LIN {X 0,Y 310.532,Z 504.322,A -85,B 0,C 180,E1 -15911.191,E2 -15911.191} C_VEL
LIN {X 0,Y 308.815,Z 514.48,A -85,B 0,C 180,E1 -15912.908,E2 -15912.908} C_VEL
LIN {X 0,Y 307.317,Z 523.179,A -85,B 0,C 180,E1 -15914.758,E2 -15914.758} C_VEL
LIN {X 0,Y 305.943,Z 530.654,A -85,B 0,C 180,E1 -15916.725,E2 -15916.725} C_VEL
LIN {X 0,Y 304.932,Z 536.676,A -85,B 0,C 180,E1 -15918.708,E2 -15918.708} C_VEL
LIN {X 0,Y 304.258,Z 541.45,A -85,B 0,C 180,E1 -15920.7,E2 -15920.7} C_VEL
LIN {X 0,Y 303.838,Z 545.114,A -85,B 0,C 180,E1 -15922.696,E2 -15922.696} C_VEL
LIN {X 0,Y 303.635,Z 547.768,A -85,B 0,C 180,E1 -15924.692,E2 -15924.692} C_VEL
LIN {X 0,Y 303.631,Z 549.032,A -85,B 0,C 180,E1 -15926.023,E2 -15926.023} C_VEL
LIN {X 0,Y 303.623,Z 549.85,A -85,B 0,C 180,E1 -15927.351,E2 -15927.351} C_VEL
LIN {X 0,Y 303.613,Z 550.259,A -85,B 0,C 180,E1 -15928.678,E2 -15928.678} C_VEL
LIN {X 0,Y 303.669,Z 550.277,A -85,B 0,C 180,E1 -15930.004,E2 -15930.004} C_VEL
LIN {X 0,Y 303.626,Z 549.898,A -85,B 0,C 180,E1 -15931.331,E2 -15931.331} C_VEL
LIN {X 0,Y 303.63,Z 549.077,A -85,B 0,C 180,E1 -15932.657,E2 -15932.657} C_VEL
LIN {X 0,Y 303.652,Z 547.834,A -85,B 0,C 180,E1 -15933.986,E2 -15933.986} C_VEL
LIN {X 0,Y 303.625,Z 545.862,A -85,B 0,C 180,E1 -15935.544,E2 -15935.544} C_VEL
LIN {X 0,Y 303.837,Z 542.819,A -85,B 0,C 180,E1 -15937.313,E2 -15937.313} C_VEL
LIN {X 0,Y 304.202,Z 538.362,A -85,B 0,C 180,E1 -15939.311,E2 -15939.311} C_VEL
LIN {X 0,Y 304.78,Z 532.679,A -85,B 0,C 180,E1 -15941.307,E2 -15941.307} C_VEL
LIN {X 0,Y 305.726,Z 525.55,A -85,B 0,C 180,E1 -15943.293,E2 -15943.293} C_VEL
LIN {X 0,Y 306.996,Z 516.63,A -85,B 0,C 180,E1 -15945.267,E2 -15945.267} C_VEL
LIN {X 0,Y 308.203,Z 507.257,A -85,B 0,C 180,E1 -15946.943,E2 -15946.943} C_VEL
LIN {X 0,Y 309.424,Z 497.348,A -85,B 0,C 180,E1 -15948.373,E2 -15948.373} C_VEL
LIN {X 0,Y 310.841,Z 486.113,A -85,B 0,C 180,E1 -15949.656,E2 -15949.656} C_VEL
LIN {X 0,Y 312.223,Z 473.536,A -85,B 0,C 180,E1 -15950.767,E2 -15950.767} C_VEL
LIN {X 0,Y 313.349,Z 460.657,A -85,B 0,C 180,E1 -15951.593,E2 -15951.593} C_VEL
LIN {X 0,Y 314.132,Z 448.168,A -85,B 0,C 180,E1 -15952.141,E2 -15952.141} C_VEL
LIN {X 0,Y 314.99,Z 419.656,A -85,B 0,C 180,E1 -15952.858,E2 -15952.858} C_VEL
LIN {X 0,Y 315.888,Z 380.038,A -85,B 0,C 180,E1 -15953.803,E2 -15953.803} C_VEL
LIN {X 0,Y 310.923,Z 346.154,A -85,B 0,C 180,E1 -15955.03,E2 -15955.03} C_VEL
LIN {X 0,Y 309.644,Z 338.018,A -85,B 0,C 180,E1 -15955.349,E2 -15955.349} C_VEL
LIN {X 0,Y 309.994,Z 334.693,A -85,B 0,C 180,E1 -15956.24,E2 -15956.24} C_VEL
LIN {X 0,Y 308.58,Z 326.696,A -85,B 0,C 180,E1 -15958.576,E2 -15958.576} C_VEL
LIN {X 0,Y 305.968,Z 314.569,A -85,B 0,C 180,E1 -15962.281,E2 -15962.281} C_VEL
LIN {X 0,Y 305.501,Z 312.43,A -85,B 0,C 180,E1 -15963.022,E2 -15963.022} C_VEL
LIN {X 0,Y 305.481,Z 312.431,A -85,B 0,C 180,E1 -15966.741,E2 -15966.741} C_VEL
LIN {X 0,Y 305.46,Z 312.438,A -85,B 0,C 180,E1 -15970.601,E2 -15970.601} C_VEL
LIN {X 0,Y 305.431,Z 312.437,A -85,B 0,C 180,E1 -15973.656,E2 -15973.656} C_VEL
LIN {X 0,Y 305.459,Z 312.433,A -85,B 0,C 180,E1 -15977.415,E2 -15977.415} C_VEL
LIN {X 0,Y 305.471,Z 312.431,A -85,B 0,C 180,E1 -15981.597,E2 -15981.597} C_VEL
LIN {X 0,Y 305.466,Z 312.435,A -85,B 0,C 180,E1 -15984.887,E2 -15984.887} C_VEL
LIN {X 0,Y 305.446,Z 312.437,A -85,B 0,C 180,E1 -15988.359,E2 -15988.359} C_VEL
LIN {X 0,Y 305.509,Z 312.43,A -85,B 0,C 180,E1 -15991.113,E2 -15991.113} C_VEL
LIN {X 0,Y 305.567,Z 312.419,A -85,B 0,C 180,E1 -15994.087,E2 -15994.087} C_VEL
LIN {X 0,Y 305.465,Z 312.433,A -85,B 0,C 180,E1 -15998.4,E2 -15998.4} C_VEL
LIN {X 0,Y 305.535,Z 312.42,A -85,B 0,C 180,E1 -16002.601,E2 -16002.601} C_VEL
LIN {X 0,Y 305.626,Z 312.412,A -85,B 0,C 180,E1 -16005.348,E2 -16005.348} C_VEL
LIN {X 0,Y 305.624,Z 312.416,A -85,B 0,C 180,E1 -16009.399,E2 -16009.399} C_VEL
LIN {X 0,Y 305.787,Z 312.391,A -85,B 0,C 180,E1 -16012.074,E2 -16012.074} C_VEL
LIN {X 0,Y 305.68,Z 312.402,A -85,B 0,C 180,E1 -16014.723,E2 -16014.723} C_VEL
LIN {X 0,Y 305.952,Z 312.362,A -85,B 0,C 180,E1 -16018.684,E2 -16018.684} C_VEL
LIN {X 0,Y 305.951,Z 312.37,A -85,B 0,C 180,E1 -16021.316,E2 -16021.316} C_VEL
LIN {X 0,Y 305.665,Z 312.409,A -85,B 0,C 180,E1 -16025.277,E2 -16025.277} C_VEL
LIN {X 0,Y 305.738,Z 312.4,A -85,B 0,C 180,E1 -16027.928,E2 -16027.928} C_VEL
LIN {X 0,Y 305.596,Z 312.419,A -85,B 0,C 180,E1 -16031.945,E2 -16031.945} C_VEL
LIN {X 0,Y 305.609,Z 312.414,A -85,B 0,C 180,E1 -16035.013,E2 -16035.013} C_VEL
LIN {X 0,Y 305.518,Z 312.422,A -85,B 0,C 180,E1 -16038.787,E2 -16038.787} C_VEL
LIN {X 0,Y 305.459,Z 312.432,A -85,B 0,C 180,E1 -16043.025,E2 -16043.025} C_VEL
LIN {X 0,Y 305.445,Z 312.437,A -85,B 0,C 180,E1 -16046.186,E2 -16046.186} C_VEL
LIN {X 0,Y 305.423,Z 312.431,A -85,B 0,C 180,E1 -16049.023,E2 -16049.023} C_VEL
LIN {X 0,Y 305.437,Z 312.427,A -85,B 0,C 180,E1 -16051.953,E2 -16051.953} C_VEL
LIN {X 0,Y 305.463,Z 312.429,A -85,B 0,C 180,E1 -16055.113,E2 -16055.113} C_VEL
LIN {X 0,Y 305.438,Z 312.44,A -85,B 0,C 180,E1 -16058.524,E2 -16058.524} C_VEL
LIN {X 0,Y 305.406,Z 312.442,A -85,B 0,C 180,E1 -16062.574,E2 -16062.574} C_VEL
LIN {X 0,Y 305.42,Z 312.441,A -85,B 0,C 180,E1 -16066.342,E2 -16066.342} C_VEL
LIN {X 0,Y 305.396,Z 312.439,A -85,B 0,C 180,E1 -16069.88,E2 -16069.88} C_VEL
LIN {X 0,Y 305.452,Z 312.433,A -85,B 0,C 180,E1 -16073.639,E2 -16073.639} C_VEL
LIN {X 0,Y 305.448,Z 312.435,A -85,B 0,C 180,E1 -16076.479,E2 -16076.479} C_VEL
LIN {X 0,Y 305.418,Z 312.439,A -85,B 0,C 180,E1 -16079.583,E2 -16079.583} C_VEL
LIN {X 0,Y 305.459,Z 312.435,A -85,B 0,C 180,E1 -16082.6,E2 -16082.6} C_VEL
LIN {X 0,Y 305.479,Z 312.431,A -85,B 0,C 180,E1 -16085.533,E2 -16085.533} C_VEL
LIN {X 0,Y 305.49,Z 312.43,A -85,B 0,C 180,E1 -16089.81,E2 -16089.81} C_VEL
LIN {X 0,Y 305.557,Z 312.421,A -85,B 0,C 180,E1 -16093.975,E2 -16093.975} C_VEL
LIN {X 0,Y 305.592,Z 312.417,A -85,B 0,C 180,E1 -16096.701,E2 -16096.701} C_VEL
LIN {X 0,Y 305.758,Z 312.399,A -85,B 0,C 180,E1 -16101.258,E2 -16101.258} C_VEL
LIN {X 0,Y 305.789,Z 312.396,A -85,B 0,C 180,E1 -16103.397,E2 -16103.397} C_VEL
LIN {X 0,Y 305.948,Z 312.372,A -85,B 0,C 180,E1 -16108.68,E2 -16108.68} C_VEL
LIN {X 0,Y 305.937,Z 312.375,A -85,B 0,C 180,E1 -16111.312,E2 -16111.312} C_VEL
LIN {X 0,Y 305.675,Z 312.496,A -85,B 0,C 180,E1 -16115.065,E2 -16115.065} C_VEL
LIN {X 0,Y 306.684,Z 317.033,A -85,B 0,C 180,E1 -16116.513,E2 -16116.513} C_VEL
LIN {X 0,Y 315.207,Z 340.384,A -85,B 0,C 180,E1 -16117.762,E2 -16117.762} C_VEL
LIN {X 0,Y 316.534,Z 347.221,A -85,B 0,C 180,E1 -16118.031,E2 -16118.031} C_VEL
LIN {X 0,Y 314.507,Z 424.142,A -85,B 0,C 180,E1 -16119.877,E2 -16119.877} C_VEL
LIN {X 0,Y 313.857,Z 437.197,A -85,B 0,C 180,E1 -16120.437,E2 -16120.437} C_VEL
LIN {X 0,Y 312.968,Z 449.965,A -85,B 0,C 180,E1 -16121.245,E2 -16121.245} C_VEL
LIN {X 0,Y 311.97,Z 461.032,A -85,B 0,C 180,E1 -16122.187,E2 -16122.187} C_VEL
LIN {X 0,Y 310.666,Z 472.181,A -85,B 0,C 180,E1 -16123.402,E2 -16123.402} C_VEL
LIN {X 0,Y 309.211,Z 483.594,A -85,B 0,C 180,E1 -16124.978,E2 -16124.978} C_VEL
LIN {X 0,Y 308.01,Z 492.9,A -85,B 0,C 180,E1 -16126.597,E2 -16126.597} C_VEL
LIN {X 0,Y 306.843,Z 501.093,A -85,B 0,C 180,E1 -16128.351,E2 -16128.351} C_VEL
LIN {X 0,Y 305.759,Z 509.186,A -85,B 0,C 180,E1 -16130.514,E2 -16130.514} C_VEL
LIN {X 0,Y 305.129,Z 514.182,A -85,B 0,C 180,E1 -16132.188,E2 -16132.188} C_VEL
LIN {X 0,Y 304.432,Z 519.747,A -85,B 0,C 180,E1 -16134.547,E2 -16134.547} C_VEL
LIN {X 0,Y 303.886,Z 523.579,A -85,B 0,C 180,E1 -16136.8,E2 -16136.8} C_VEL
LIN {X 0,Y 303.543,Z 526.171,A -85,B 0,C 180,E1 -16139.085,E2 -16139.085} C_VEL
LIN {X 0,Y 303.425,Z 527.406,A -85,B 0,C 180,E1 -16141.018,E2 -16141.018} C_VEL
LIN {X 0,Y 303.471,Z 527.743,A -85,B 0,C 180,E1 -16143.517,E2 -16143.517} C_VEL
LIN {X 0,Y 303.709,Z 526.753,A -85,B 0,C 180,E1 -16145.912,E2 -16145.912} C_VEL
LIN {X 0,Y 304.143,Z 524.521,A -85,B 0,C 180,E1 -16148.218,E2 -16148.218} C_VEL
LIN {X 0,Y 304.8,Z 521.115,A -85,B 0,C 180,E1 -16150.456,E2 -16150.456} C_VEL
LIN {X 0,Y 305.637,Z 516.547,A -85,B 0,C 180,E1 -16152.623,E2 -16152.623} C_VEL
LIN {X 0,Y 306.766,Z 510.68,A -85,B 0,C 180,E1 -16154.748,E2 -16154.748} C_VEL
LIN {X 0,Y 308.203,Z 503.227,A -85,B 0,C 180,E1 -16156.851,E2 -16156.851} C_VEL
LIN {X 0,Y 309.972,Z 493.999,A -85,B 0,C 180,E1 -16158.889,E2 -16158.889} C_VEL
LIN {X 0,Y 311.555,Z 484.866,A -85,B 0,C 180,E1 -16160.507,E2 -16160.507} C_VEL
LIN {X 0,Y 312.9,Z 475.839,A -85,B 0,C 180,E1 -16161.814,E2 -16161.814} C_VEL
LIN {X 0,Y 314.575,Z 464.879,A -85,B 0,C 180,E1 -16163.071,E2 -16163.071} C_VEL
LIN {X 0,Y 315.779,Z 454.371,A -85,B 0,C 180,E1 -16164.041,E2 -16164.041} C_VEL
LIN {X 0,Y 316.943,Z 441.922,A -85,B 0,C 180,E1 -16164.915,E2 -16164.915} C_VEL
LIN {X 0,Y 317.748,Z 429.439,A -85,B 0,C 180,E1 -16165.534,E2 -16165.534} C_VEL
LIN {X 0,Y 317.977,Z 425.769,A -85,B 0,C 180,E1 -16165.662,E2 -16165.662} C_VEL
LIN {X 0,Y 317.615,Z 420.025,A -85,B 0,C 180,E1 -16165.907,E2 -16165.907} C_VEL
LIN {X 0,Y 313.109,Z 401.411,A -85,B 0,C 180,E1 -16166.843,E2 -16166.843} C_VEL
LIN {X 0,Y 312.707,Z 395.612,A -85,B 0,C 180,E1 -16167.035,E2 -16167.035} C_VEL
LIN {X 0,Y 314.177,Z 349.617,A -85,B 0,C 180,E1 -16168.164,E2 -16168.164} C_VEL
LIN {X 0,Y 308.843,Z 336.559,A -85,B 0,C 180,E1 -16169.123,E2 -16169.123} C_VEL
LIN {X 0,Y 301.142,Z 320.791,A -85,B 0,C 180,E1 -16170.507,E2 -16170.507} C_VEL
LIN {X 0,Y 299.59,Z 317.573,A -85,B 0,C 180,E1 -16170.823,E2 -16170.823} C_VEL
LIN {X 0,Y 298.45,Z 313.316,A -85,B 0,C 180,E1 -16172.38,E2 -16172.38} C_VEL
LIN {X 0,Y 298.445,Z 313.316,A -85,B 0,C 180,E1 -16174.92,E2 -16174.92} C_VEL
LIN {X 0,Y 298.397,Z 313.319,A -85,B 0,C 180,E1 -16179.311,E2 -16179.311} C_VEL
LIN {X 0,Y 298.491,Z 313.306,A -85,B 0,C 180,E1 -16182.176,E2 -16182.176} C_VEL
LIN {X 0,Y 298.545,Z 313.299,A -85,B 0,C 180,E1 -16184.992,E2 -16184.992} C_VEL
LIN {X 0,Y 298.539,Z 313.292,A -85,B 0,C 180,E1 -16189.145,E2 -16189.145} C_VEL
LIN {X 0,Y 298.688,Z 313.277,A -85,B 0,C 180,E1 -16191.884,E2 -16191.884} C_VEL
LIN {X 0,Y 298.611,Z 313.29,A -85,B 0,C 180,E1 -16194.598,E2 -16194.598} C_VEL
LIN {X 0,Y 298.879,Z 313.252,A -85,B 0,C 180,E1 -16198.653,E2 -16198.653} C_VEL
LIN {X 0,Y 298.879,Z 313.255,A -85,B 0,C 180,E1 -16201.347,E2 -16201.347} C_VEL
LIN {X 0,Y 298.745,Z 313.268,A -85,B 0,C 180,E1 -16206.755,E2 -16206.755} C_VEL
LIN {X 0,Y 298.638,Z 313.286,A -85,B 0,C 180,E1 -16209.482,E2 -16209.482} C_VEL
LIN {X 0,Y 298.507,Z 313.301,A -85,B 0,C 180,E1 -16213.617,E2 -16213.617} C_VEL
LIN {X 0,Y 298.504,Z 313.29,A -85,B 0,C 180,E1 -16216.411,E2 -16216.411} C_VEL
LIN {X 0,Y 298.494,Z 313.293,A -85,B 0,C 180,E1 -16219.669,E2 -16219.669} C_VEL
LIN {X 0,Y 298.437,Z 313.301,A -85,B 0,C 180,E1 -16223.599,E2 -16223.599} C_VEL
LIN {X 0,Y 298.453,Z 313.305,A -85,B 0,C 180,E1 -16226.578,E2 -16226.578} C_VEL
LIN {X 0,Y 298.384,Z 313.315,A -85,B 0,C 180,E1 -16229.645,E2 -16229.645} C_VEL
LIN {X 0,Y 298.362,Z 313.316,A -85,B 0,C 180,E1 -16232.804,E2 -16232.804} C_VEL
LIN {X 0,Y 298.457,Z 313.308,A -85,B 0,C 180,E1 -16236.823,E2 -16236.823} C_VEL
LIN {X 0,Y 298.428,Z 313.311,A -85,B 0,C 180,E1 -16241.108,E2 -16241.108} C_VEL
LIN {X 0,Y 298.463,Z 313.314,A -85,B 0,C 180,E1 -16245.066,E2 -16245.066} C_VEL
LIN {X 0,Y 298.43,Z 313.315,A -85,B 0,C 180,E1 -16248.903,E2 -16248.903} C_VEL
LIN {X 0,Y 298.449,Z 313.306,A -85,B 0,C 180,E1 -16253.192,E2 -16253.192} C_VEL
LIN {X 0,Y 298.453,Z 313.458,A -85,B 0,C 180,E1 -16254.395,E2 -16254.395} C_VEL
LIN {X 0,Y 301.098,Z 323.779,A -85,B 0,C 180,E1 -16257.934,E2 -16257.934} C_VEL
LIN {X 0,Y 303.507,Z 334.535,A -85,B 0,C 180,E1 -16261.363,E2 -16261.363} C_VEL
LIN {X 0,Y 303.784,Z 335.948,A -85,B 0,C 180,E1 -16261.77,E2 -16261.77} C_VEL
LIN {X 0,Y 306.903,Z 343.742,A -85,B 0,C 180,E1 -16262.363,E2 -16262.363} C_VEL
LIN {X 0,Y 311.12,Z 366.166,A -85,B 0,C 180,E1 -16263.476,E2 -16263.476} C_VEL
LIN {X 0,Y 313.3,Z 382.701,A -85,B 0,C 180,E1 -16264.165,E2 -16264.165} C_VEL
LIN {X 0,Y 311.187,Z 445.435,A -85,B 0,C 180,E1 -16265.72,E2 -16265.72} C_VEL
LIN {X 0,Y 310.209,Z 458.829,A -85,B 0,C 180,E1 -16266.294,E2 -16266.294} C_VEL
LIN {X 0,Y 308.892,Z 471.237,A -85,B 0,C 180,E1 -16267.075,E2 -16267.075} C_VEL
LIN {X 0,Y 307.374,Z 482.408,A -85,B 0,C 180,E1 -16268.018,E2 -16268.018} C_VEL
LIN {X 0,Y 305.621,Z 494.017,A -85,B 0,C 180,E1 -16269.301,E2 -16269.301} C_VEL
LIN {X 0,Y 303.838,Z 504.506,A -85,B 0,C 180,E1 -16270.761,E2 -16270.761} C_VEL
LIN {X 0,Y 302.116,Z 514.002,A -85,B 0,C 180,E1 -16272.403,E2 -16272.403} C_VEL
LIN {X 0,Y 300.442,Z 523.19,A -85,B 0,C 180,E1 -16274.4,E2 -16274.4} C_VEL
LIN {X 0,Y 299.009,Z 530.619,A -85,B 0,C 180,E1 -16276.411,E2 -16276.411} C_VEL
LIN {X 0,Y 297.924,Z 536.598,A -85,B 0,C 180,E1 -16278.438,E2 -16278.438} C_VEL
LIN {X 0,Y 297.229,Z 541.333,A -85,B 0,C 180,E1 -16280.478,E2 -16280.478} C_VEL
LIN {X 0,Y 296.786,Z 544.96,A -85,B 0,C 180,E1 -16282.521,E2 -16282.521} C_VEL
LIN {X 0,Y 296.55,Z 547.576,A -85,B 0,C 180,E1 -16284.565,E2 -16284.565} C_VEL
LIN {X 0,Y 296.528,Z 548.815,A -85,B 0,C 180,E1 -16285.927,E2 -16285.927} C_VEL
LIN {X 0,Y 296.548,Z 549.607,A -85,B 0,C 180,E1 -16287.288,E2 -16287.288} C_VEL
LIN {X 0,Y 296.53,Z 550,A -85,B 0,C 180,E1 -16288.646,E2 -16288.646} C_VEL
LIN {X 0,Y 296.581,Z 550.004,A -85,B 0,C 180,E1 -16290.004,E2 -16290.004} C_VEL
LIN {X 0,Y 296.542,Z 549.604,A -85,B 0,C 180,E1 -16291.362,E2 -16291.362} C_VEL
LIN {X 0,Y 296.555,Z 548.757,A -85,B 0,C 180,E1 -16292.721,E2 -16292.721} C_VEL
LIN {X 0,Y 296.566,Z 547.498,A -85,B 0,C 180,E1 -16294.081,E2 -16294.081} C_VEL
LIN {X 0,Y 296.574,Z 544.796,A -85,B 0,C 180,E1 -16296.125,E2 -16296.125} C_VEL
LIN {X 0,Y 296.878,Z 541.05,A -85,B 0,C 180,E1 -16298.17,E2 -16298.17} C_VEL
LIN {X 0,Y 297.346,Z 536.154,A -85,B 0,C 180,E1 -16300.214,E2 -16300.214} C_VEL
LIN {X 0,Y 298.049,Z 529.959,A -85,B 0,C 180,E1 -16302.256,E2 -16302.256} C_VEL
LIN {X 0,Y 299.19,Z 522.25,A -85,B 0,C 180,E1 -16304.283,E2 -16304.283} C_VEL
LIN {X 0,Y 300.333,Z 514.337,A -85,B 0,C 180,E1 -16305.963,E2 -16305.963} C_VEL
LIN {X 0,Y 301.559,Z 504.648,A -85,B 0,C 180,E1 -16307.639,E2 -16307.639} C_VEL
LIN {X 0,Y 303.043,Z 493.923,A -85,B 0,C 180,E1 -16309.125,E2 -16309.125} C_VEL
LIN {X 0,Y 304.318,Z 483.564,A -85,B 0,C 180,E1 -16310.271,E2 -16310.271} C_VEL
LIN {X 0,Y 305.655,Z 471.217,A -85,B 0,C 180,E1 -16311.323,E2 -16311.323} C_VEL
LIN {X 0,Y 306.839,Z 457.559,A -85,B 0,C 180,E1 -16312.164,E2 -16312.164} C_VEL
LIN {X 0,Y 307.587,Z 444.598,A -85,B 0,C 180,E1 -16312.682,E2 -16312.682} C_VEL
LIN {X 0,Y 309.249,Z 381.078,A -85,B 0,C 180,E1 -16314.236,E2 -16314.236} C_VEL
LIN {X 0,Y 304.445,Z 347.745,A -85,B 0,C 180,E1 -16315.47,E2 -16315.47} C_VEL
LIN {X 0,Y 302.859,Z 337.766,A -85,B 0,C 180,E1 -16315.876,E2 -16315.876} C_VEL
LIN {X 0,Y 302.829,Z 334.116,A -85,B 0,C 180,E1 -16316.91,E2 -16316.91} C_VEL
LIN {X 0,Y 300.678,Z 323.498,A -85,B 0,C 180,E1 -16320.136,E2 -16320.136} C_VEL
LIN {X 0,Y 298.446,Z 313.31,A -85,B 0,C 180,E1 -16323.401,E2 -16323.401} C_VEL
LIN {X 0,Y 298.452,Z 313.307,A -85,B 0,C 180,E1 -16326.809,E2 -16326.809} C_VEL
LIN {X 0,Y 298.393,Z 313.316,A -85,B 0,C 180,E1 -16331.089,E2 -16331.089} C_VEL
LIN {X 0,Y 298.405,Z 313.312,A -85,B 0,C 180,E1 -16333.104,E2 -16333.104} C_VEL
LIN {X 0,Y 298.409,Z 313.314,A -85,B 0,C 180,E1 -16336.922,E2 -16336.922} C_VEL
LIN {X 0,Y 298.403,Z 313.314,A -85,B 0,C 180,E1 -16341.009,E2 -16341.009} C_VEL
LIN {X 0,Y 298.41,Z 313.312,A -85,B 0,C 180,E1 -16343.929,E2 -16343.929} C_VEL
LIN {X 0,Y 298.397,Z 313.315,A -85,B 0,C 180,E1 -16347.2,E2 -16347.2} C_VEL
LIN {X 0,Y 298.457,Z 313.305,A -85,B 0,C 180,E1 -16351.904,E2 -16351.904} C_VEL
LIN {X 0,Y 298.484,Z 313.305,A -85,B 0,C 180,E1 -16354.924,E2 -16354.924} C_VEL
LIN {X 0,Y 298.42,Z 313.311,A -85,B 0,C 180,E1 -16359.313,E2 -16359.313} C_VEL
LIN {X 0,Y 298.466,Z 313.299,A -85,B 0,C 180,E1 -16362.175,E2 -16362.175} C_VEL
LIN {X 0,Y 298.589,Z 313.284,A -85,B 0,C 180,E1 -16364.995,E2 -16364.995} C_VEL
LIN {X 0,Y 298.583,Z 313.293,A -85,B 0,C 180,E1 -16369.146,E2 -16369.146} C_VEL
LIN {X 0,Y 298.733,Z 313.27,A -85,B 0,C 180,E1 -16371.885,E2 -16371.885} C_VEL
LIN {X 0,Y 298.651,Z 313.277,A -85,B 0,C 180,E1 -16374.599,E2 -16374.599} C_VEL
LIN {X 0,Y 298.919,Z 313.236,A -85,B 0,C 180,E1 -16378.653,E2 -16378.653} C_VEL
LIN {X 0,Y 298.918,Z 313.245,A -85,B 0,C 180,E1 -16381.347,E2 -16381.347} C_VEL
LIN {X 0,Y 298.634,Z 313.286,A -85,B 0,C 180,E1 -16385.402,E2 -16385.402} C_VEL
LIN {X 0,Y 298.684,Z 313.277,A -85,B 0,C 180,E1 -16388.116,E2 -16388.116} C_VEL
LIN {X 0,Y 298.548,Z 313.294,A -85,B 0,C 180,E1 -16392.232,E2 -16392.232} C_VEL
LIN {X 0,Y 298.549,Z 313.294,A -85,B 0,C 180,E1 -16395.166,E2 -16395.166} C_VEL
LIN {X 0,Y 298.443,Z 313.305,A -85,B 0,C 180,E1 -16399.616,E2 -16399.616} C_VEL
LIN {X 0,Y 298.388,Z 313.315,A -85,B 0,C 180,E1 -16403.604,E2 -16403.604} C_VEL
LIN {X 0,Y 298.401,Z 313.31,A -85,B 0,C 180,E1 -16406.583,E2 -16406.583} C_VEL
LIN {X 0,Y 298.357,Z 313.311,A -85,B 0,C 180,E1 -16409.648,E2 -16409.648} C_VEL
LIN {X 0,Y 298.394,Z 313.306,A -85,B 0,C 180,E1 -16412.8,E2 -16412.8} C_VEL
LIN {X 0,Y 298.406,Z 313.311,A -85,B 0,C 180,E1 -16416.072,E2 -16416.072} C_VEL
LIN {X 0,Y 298.348,Z 313.318,A -85,B 0,C 180,E1 -16419.496,E2 -16419.496} C_VEL
LIN {X 0,Y 298.372,Z 313.315,A -85,B 0,C 180,E1 -16423.096,E2 -16423.096} C_VEL
LIN {X 0,Y 298.374,Z 313.318,A -85,B 0,C 180,E1 -16426.913,E2 -16426.913} C_VEL
LIN {X 0,Y 298.367,Z 313.319,A -85,B 0,C 180,E1 -16431.015,E2 -16431.015} C_VEL
LIN {X 0,Y 298.394,Z 313.313,A -85,B 0,C 180,E1 -16433.924,E2 -16433.924} C_VEL
LIN {X 0,Y 298.384,Z 313.317,A -85,B 0,C 180,E1 -16437.196,E2 -16437.196} C_VEL
LIN {X 0,Y 298.374,Z 313.319,A -85,B 0,C 180,E1 -16440.635,E2 -16440.635} C_VEL
LIN {X 0,Y 298.444,Z 313.313,A -85,B 0,C 180,E1 -16444.917,E2 -16444.917} C_VEL
LIN {X 0,Y 298.407,Z 313.313,A -85,B 0,C 180,E1 -16447.86,E2 -16447.86} C_VEL
LIN {X 0,Y 298.471,Z 313.306,A -85,B 0,C 180,E1 -16450.749,E2 -16450.749} C_VEL
LIN {X 0,Y 298.592,Z 313.291,A -85,B 0,C 180,E1 -16454.991,E2 -16454.991} C_VEL
LIN {X 0,Y 298.588,Z 313.292,A -85,B 0,C 180,E1 -16459.143,E2 -16459.143} C_VEL
LIN {X 0,Y 298.702,Z 313.276,A -85,B 0,C 180,E1 -16461.881,E2 -16461.881} C_VEL
LIN {X 0,Y 298.63,Z 313.284,A -85,B 0,C 180,E1 -16464.594,E2 -16464.594} C_VEL
LIN {X 0,Y 298.914,Z 313.248,A -85,B 0,C 180,E1 -16468.648,E2 -16468.648} C_VEL
LIN {X 0,Y 298.905,Z 313.251,A -85,B 0,C 180,E1 -16471.343,E2 -16471.343} C_VEL
LIN {X 0,Y 298.612,Z 313.39,A -85,B 0,C 180,E1 -16474.678,E2 -16474.678} C_VEL
LIN {X 0,Y 299.557,Z 317.277,A -85,B 0,C 180,E1 -16475.95,E2 -16475.95} C_VEL
LIN {X 0,Y 308.309,Z 341.137,A -85,B 0,C 180,E1 -16477.279,E2 -16477.279} C_VEL
LIN {X 0,Y 309.872,Z 347.843,A -85,B 0,C 180,E1 -16477.57,E2 -16477.57} C_VEL
LIN {X 0,Y 307.812,Z 424.3,A -85,B 0,C 180,E1 -16479.447,E2 -16479.447} C_VEL
LIN {X 0,Y 307.155,Z 437.346,A -85,B 0,C 180,E1 -16480.017,E2 -16480.017} C_VEL
LIN {X 0,Y 306.243,Z 449.928,A -85,B 0,C 180,E1 -16480.825,E2 -16480.825} C_VEL
LIN {X 0,Y 305.216,Z 461.07,A -85,B 0,C 180,E1 -16481.787,E2 -16481.787} C_VEL
LIN {X 0,Y 303.861,Z 472.273,A -85,B 0,C 180,E1 -16483.027,E2 -16483.027} C_VEL
LIN {X 0,Y 302.362,Z 483.606,A -85,B 0,C 180,E1 -16484.619,E2 -16484.619} C_VEL
LIN {X 0,Y 301.111,Z 492.907,A -85,B 0,C 180,E1 -16486.259,E2 -16486.259} C_VEL
LIN {X 0,Y 299.879,Z 501.279,A -85,B 0,C 180,E1 -16488.085,E2 -16488.085} C_VEL
LIN {X 0,Y 298.798,Z 509.117,A -85,B 0,C 180,E1 -16490.217,E2 -16490.217} C_VEL
LIN {X 0,Y 298.032,Z 514.805,A -85,B 0,C 180,E1 -16492.16,E2 -16492.16} C_VEL
LIN {X 0,Y 297.374,Z 519.977,A -85,B 0,C 180,E1 -16494.424,E2 -16494.424} C_VEL
LIN {X 0,Y 296.815,Z 523.819,A -85,B 0,C 180,E1 -16496.729,E2 -16496.729} C_VEL
LIN {X 0,Y 296.48,Z 526.114,A -85,B 0,C 180,E1 -16498.708,E2 -16498.708} C_VEL
LIN {X 0,Y 296.333,Z 527.815,A -85,B 0,C 180,E1 -16501.443,E2 -16501.443} C_VEL
LIN {X 0,Y 296.395,Z 527.982,A -85,B 0,C 180,E1 -16503.91,E2 -16503.91} C_VEL
LIN {X 0,Y 296.68,Z 526.817,A -85,B 0,C 180,E1 -16506.349,E2 -16506.349} C_VEL
LIN {X 0,Y 297.183,Z 524.453,A -85,B 0,C 180,E1 -16508.702,E2 -16508.702} C_VEL
LIN {X 0,Y 297.922,Z 520.922,A -85,B 0,C 180,E1 -16510.985,E2 -16510.985} C_VEL
LIN {X 0,Y 298.81,Z 516.249,A -85,B 0,C 180,E1 -16513.187,E2 -16513.187} C_VEL
LIN {X 0,Y 300.062,Z 510.211,A -85,B 0,C 180,E1 -16515.359,E2 -16515.359} C_VEL
LIN {X 0,Y 301.62,Z 502.588,A -85,B 0,C 180,E1 -16517.489,E2 -16517.489} C_VEL
LIN {X 0,Y 303.206,Z 494.727,A -85,B 0,C 180,E1 -16519.253,E2 -16519.253} C_VEL
LIN {X 0,Y 304.771,Z 486.159,A -85,B 0,C 180,E1 -16520.829,E2 -16520.829} C_VEL
LIN {X 0,Y 306.257,Z 476.906,A -85,B 0,C 180,E1 -16522.226,E2 -16522.226} C_VEL
LIN {X 0,Y 307.932,Z 466.519,A -85,B 0,C 180,E1 -16523.477,E2 -16523.477} C_VEL
LIN {X 0,Y 309.185,Z 456.404,A -85,B 0,C 180,E1 -16524.461,E2 -16524.461} C_VEL
LIN {X 0,Y 310.455,Z 443.807,A -85,B 0,C 180,E1 -16525.394,E2 -16525.394} C_VEL
LIN {X 0,Y 311.344,Z 431.002,A -85,B 0,C 180,E1 -16526.073,E2 -16526.073} C_VEL
LIN {X 0,Y 312.029,Z 417.729,A -85,B 0,C 180,E1 -16526.493,E2 -16526.493} C_VEL
LIN {X 0,Y 312.707,Z 395.612,A -85,B 0,C 180,E1 -16527.035,E2 -16527.035} C_VEL
LIN {X 0,Y 312.314,Z 389.817,A -85,B 0,C 180,E1 -16527.236,E2 -16527.236} C_VEL
LIN {X 0,Y 307.946,Z 371.209,A -85,B 0,C 180,E1 -16528.222,E2 -16528.222} C_VEL
LIN {X 0,Y 307.614,Z 365.414,A -85,B 0,C 180,E1 -16528.425,E2 -16528.425} C_VEL
LIN {X 0,Y 308.102,Z 351.664,A -85,B 0,C 180,E1 -16528.769,E2 -16528.769} C_VEL
LIN {X 0,Y 302.709,Z 338.584,A -85,B 0,C 180,E1 -16529.778,E2 -16529.778} C_VEL
LIN {X 0,Y 295.398,Z 323.718,A -85,B 0,C 180,E1 -16531.149,E2 -16531.149} C_VEL
LIN {X 0,Y 292.402,Z 317.923,A -85,B 0,C 180,E1 -16531.758,E2 -16531.758} C_VEL
LIN {X 0,Y 291.416,Z 314.191,A -85,B 0,C 180,E1 -16533.148,E2 -16533.148} C_VEL
LIN {X 0,Y 291.336,Z 314.202,A -85,B 0,C 180,E1 -16537.296,E2 -16537.296} C_VEL
LIN {X 0,Y 291.419,Z 314.191,A -85,B 0,C 180,E1 -16540.267,E2 -16540.267} C_VEL
LIN {X 0,Y 291.475,Z 314.178,A -85,B 0,C 180,E1 -16544.65,E2 -16544.65} C_VEL
LIN {X 0,Y 291.485,Z 314.172,A -85,B 0,C 180,E1 -16548.879,E2 -16548.879} C_VEL
LIN {X 0,Y 291.636,Z 314.156,A -85,B 0,C 180,E1 -16551.686,E2 -16551.686} C_VEL
LIN {X 0,Y 291.582,Z 314.165,A -85,B 0,C 180,E1 -16554.467,E2 -16554.467} C_VEL
LIN {X 0,Y 291.845,Z 314.128,A -85,B 0,C 180,E1 -16558.62,E2 -16558.62} C_VEL
LIN {X 0,Y 291.845,Z 314.131,A -85,B 0,C 180,E1 -16561.38,E2 -16561.38} C_VEL
LIN {X 0,Y 291.695,Z 314.144,A -85,B 0,C 180,E1 -16566.919,E2 -16566.919} C_VEL
LIN {X 0,Y 291.587,Z 314.164,A -85,B 0,C 180,E1 -16569.713,E2 -16569.713} C_VEL
LIN {X 0,Y 291.476,Z 314.176,A -85,B 0,C 180,E1 -16573.953,E2 -16573.953} C_VEL
LIN {X 0,Y 291.439,Z 314.178,A -85,B 0,C 180,E1 -16578.27,E2 -16578.27} C_VEL
LIN {X 0,Y 291.367,Z 314.18,A -85,B 0,C 180,E1 -16581.212,E2 -16581.212} C_VEL
LIN {X 0,Y 291.392,Z 314.175,A -85,B 0,C 180,E1 -16584.206,E2 -16584.206} C_VEL
LIN {X 0,Y 291.386,Z 314.183,A -85,B 0,C 180,E1 -16587.275,E2 -16587.275} C_VEL
LIN {X 0,Y 291.301,Z 314.197,A -85,B 0,C 180,E1 -16590.441,E2 -16590.441} C_VEL
LIN {X 0,Y 291.315,Z 314.199,A -85,B 0,C 180,E1 -16593.702,E2 -16593.702} C_VEL
LIN {X 0,Y 291.395,Z 314.189,A -85,B 0,C 180,E1 -16597.272,E2 -16597.272} C_VEL
LIN {X 0,Y 291.38,Z 314.19,A -85,B 0,C 180,E1 -16600.635,E2 -16600.635} C_VEL
LIN {X 0,Y 291.38,Z 314.194,A -85,B 0,C 180,E1 -16604.385,E2 -16604.385} C_VEL
LIN {X 0,Y 291.365,Z 314.194,A -85,B 0,C 180,E1 -16608.396,E2 -16608.396} C_VEL
LIN {X 0,Y 291.363,Z 314.195,A -85,B 0,C 180,E1 -16611.169,E2 -16611.169} C_VEL
LIN {X 0,Y 291.405,Z 314.266,A -85,B 0,C 180,E1 -16613.574,E2 -16613.574} C_VEL
LIN {X 0,Y 294.031,Z 324.386,A -85,B 0,C 180,E1 -16617.197,E2 -16617.197} C_VEL
LIN {X 0,Y 296.598,Z 335.614,A -85,B 0,C 180,E1 -16620.872,E2 -16620.872} C_VEL
LIN {X 0,Y 301.111,Z 346.332,A -85,B 0,C 180,E1 -16621.761,E2 -16621.761} C_VEL
LIN {X 0,Y 305.102,Z 368.038,A -85,B 0,C 180,E1 -16622.867,E2 -16622.867} C_VEL
LIN {X 0,Y 307.089,Z 383.433,A -85,B 0,C 180,E1 -16623.535,E2 -16623.535} C_VEL
LIN {X 0,Y 304.934,Z 445.056,A -85,B 0,C 180,E1 -16625.095,E2 -16625.095} C_VEL
LIN {X 0,Y 303.908,Z 458.523,A -85,B 0,C 180,E1 -16625.681,E2 -16625.681} C_VEL
LIN {X 0,Y 302.551,Z 470.934,A -85,B 0,C 180,E1 -16626.475,E2 -16626.475} C_VEL
LIN {X 0,Y 300.84,Z 482.901,A -85,B 0,C 180,E1 -16627.515,E2 -16627.515} C_VEL
LIN {X 0,Y 299.018,Z 494.371,A -85,B 0,C 180,E1 -16628.822,E2 -16628.822} C_VEL
LIN {X 0,Y 297.162,Z 504.756,A -85,B 0,C 180,E1 -16630.311,E2 -16630.311} C_VEL
LIN {X 0,Y 295.36,Z 514.132,A -85,B 0,C 180,E1 -16631.987,E2 -16631.987} C_VEL
LIN {X 0,Y 293.579,Z 523.23,A -85,B 0,C 180,E1 -16634.026,E2 -16634.026} C_VEL
LIN {X 0,Y 292.09,Z 530.592,A -85,B 0,C 180,E1 -16636.083,E2 -16636.083} C_VEL
LIN {X 0,Y 290.935,Z 536.519,A -85,B 0,C 180,E1 -16638.157,E2 -16638.157} C_VEL
LIN {X 0,Y 290.185,Z 541.214,A -85,B 0,C 180,E1 -16640.245,E2 -16640.245} C_VEL
LIN {X 0,Y 289.716,Z 544.806,A -85,B 0,C 180,E1 -16642.338,E2 -16642.338} C_VEL
LIN {X 0,Y 289.473,Z 547.481,A -85,B 0,C 180,E1 -16644.518,E2 -16644.518} C_VEL
LIN {X 0,Y 289.43,Z 548.596,A -85,B 0,C 180,E1 -16645.827,E2 -16645.827} C_VEL
LIN {X 0,Y 289.473,Z 549.367,A -85,B 0,C 180,E1 -16647.222,E2 -16647.222} C_VEL
LIN {X 0,Y 289.45,Z 549.743,A -85,B 0,C 180,E1 -16648.613,E2 -16648.613} C_VEL
LIN {X 0,Y 289.495,Z 549.729,A -85,B 0,C 180,E1 -16650.005,E2 -16650.005} C_VEL
LIN {X 0,Y 289.461,Z 549.299,A -85,B 0,C 180,E1 -16651.396,E2 -16651.396} C_VEL
LIN {X 0,Y 289.482,Z 548.428,A -85,B 0,C 180,E1 -16652.787,E2 -16652.787} C_VEL
LIN {X 0,Y 289.464,Z 547.148,A -85,B 0,C 180,E1 -16654.181,E2 -16654.181} C_VEL
LIN {X 0,Y 289.498,Z 544.405,A -85,B 0,C 180,E1 -16656.276,E2 -16656.276} C_VEL
LIN {X 0,Y 289.833,Z 540.618,A -85,B 0,C 180,E1 -16658.37,E2 -16658.37} C_VEL
LIN {X 0,Y 290.322,Z 535.674,A -85,B 0,C 180,E1 -16660.464,E2 -16660.464} C_VEL
LIN {X 0,Y 291.08,Z 529.428,A -85,B 0,C 180,E1 -16662.554,E2 -16662.554} C_VEL
LIN {X 0,Y 292.226,Z 521.633,A -85,B 0,C 180,E1 -16664.63,E2 -16664.63} C_VEL
LIN {X 0,Y 293.453,Z 513.641,A -85,B 0,C 180,E1 -16666.348,E2 -16666.348} C_VEL
LIN {X 0,Y 294.732,Z 503.863,A -85,B 0,C 180,E1 -16668.062,E2 -16668.062} C_VEL
LIN {X 0,Y 296.265,Z 493.028,A -85,B 0,C 180,E1 -16669.58,E2 -16669.58} C_VEL
LIN {X 0,Y 297.647,Z 482.506,A -85,B 0,C 180,E1 -16670.746,E2 -16670.746} C_VEL
LIN {X 0,Y 299.062,Z 469.876,A -85,B 0,C 180,E1 -16671.817,E2 -16671.817} C_VEL
LIN {X 0,Y 300.174,Z 456.583,A -85,B 0,C 180,E1 -16672.638,E2 -16672.638} C_VEL
LIN {X 0,Y 300.969,Z 443.009,A -85,B 0,C 180,E1 -16673.164,E2 -16673.164} C_VEL
LIN {X 0,Y 302.525,Z 380.928,A -85,B 0,C 180,E1 -16674.721,E2 -16674.721} C_VEL
LIN {X 0,Y 297.844,Z 348.646,A -85,B 0,C 180,E1 -16675.958,E2 -16675.958} C_VEL
LIN {X 0,Y 296.054,Z 337.468,A -85,B 0,C 180,E1 -16676.436,E2 -16676.436} C_VEL
LIN {X 0,Y 294.991,Z 330.809,A -85,B 0,C 180,E1 -16678.459,E2 -16678.459} C_VEL
LIN {X 0,Y 292.17,Z 317.667,A -85,B 0,C 180,E1 -16682.658,E2 -16682.658} C_VEL
LIN {X 0,Y 291.415,Z 314.188,A -85,B 0,C 180,E1 -16683.843,E2 -16683.843} C_VEL
LIN {X 0,Y 291.382,Z 314.187,A -85,B 0,C 180,E1 -16687.255,E2 -16687.255} C_VEL
LIN {X 0,Y 291.339,Z 314.197,A -85,B 0,C 180,E1 -16690.644,E2 -16690.644} C_VEL
LIN {X 0,Y 291.297,Z 314.203,A -85,B 0,C 180,E1 -16694.403,E2 -16694.403} C_VEL
LIN {X 0,Y 291.332,Z 314.198,A -85,B 0,C 180,E1 -16698.405,E2 -16698.405} C_VEL
LIN {X 0,Y 291.351,Z 314.191,A -85,B 0,C 180,E1 -16701.158,E2 -16701.158} C_VEL
LIN {X 0,Y 291.36,Z 314.194,A -85,B 0,C 180,E1 -16704.626,E2 -16704.626} C_VEL
LIN {X 0,Y 291.37,Z 314.189,A -85,B 0,C 180,E1 -16707.95,E2 -16707.95} C_VEL
LIN {X 0,Y 291.376,Z 314.19,A -85,B 0,C 180,E1 -16711.158,E2 -16711.158} C_VEL
LIN {X 0,Y 291.414,Z 314.183,A -85,B 0,C 180,E1 -16714.272,E2 -16714.272} C_VEL
LIN {X 0,Y 291.372,Z 314.19,A -85,B 0,C 180,E1 -16717.299,E2 -16717.299} C_VEL
LIN {X 0,Y 291.394,Z 314.183,A -85,B 0,C 180,E1 -16720.266,E2 -16720.266} C_VEL
LIN {X 0,Y 291.501,Z 314.163,A -85,B 0,C 180,E1 -16724.666,E2 -16724.666} C_VEL
LIN {X 0,Y 291.529,Z 314.169,A -85,B 0,C 180,E1 -16728.88,E2 -16728.88} C_VEL
LIN {X 0,Y 291.681,Z 314.15,A -85,B 0,C 180,E1 -16731.688,E2 -16731.688} C_VEL
LIN {X 0,Y 291.622,Z 314.152,A -85,B 0,C 180,E1 -16734.468,E2 -16734.468} C_VEL
LIN {X 0,Y 291.886,Z 314.11,A -85,B 0,C 180,E1 -16738.62,E2 -16738.62} C_VEL
LIN {X 0,Y 291.885,Z 314.121,A -85,B 0,C 180,E1 -16741.38,E2 -16741.38} C_VEL
LIN {X 0,Y 291.645,Z 314.153,A -85,B 0,C 180,E1 -16746.541,E2 -16746.541} C_VEL
LIN {X 0,Y 291.565,Z 314.165,A -85,B 0,C 180,E1 -16749.714,E2 -16749.714} C_VEL
LIN {X 0,Y 291.515,Z 314.174,A -85,B 0,C 180,E1 -16753.951,E2 -16753.951} C_VEL
LIN {X 0,Y 291.429,Z 314.179,A -85,B 0,C 180,E1 -16756.821,E2 -16756.821} C_VEL
LIN {X 0,Y 291.395,Z 314.184,A -85,B 0,C 180,E1 -16759.842,E2 -16759.842} C_VEL
LIN {X 0,Y 291.332,Z 314.195,A -85,B 0,C 180,E1 -16764.211,E2 -16764.211} C_VEL
LIN {X 0,Y 291.329,Z 314.189,A -85,B 0,C 180,E1 -16767.281,E2 -16767.281} C_VEL
LIN {X 0,Y 291.302,Z 314.184,A -85,B 0,C 180,E1 -16770.441,E2 -16770.441} C_VEL
LIN {X 0,Y 291.346,Z 314.183,A -85,B 0,C 180,E1 -16773.698,E2 -16773.698} C_VEL
LIN {X 0,Y 291.351,Z 314.189,A -85,B 0,C 180,E1 -16777.245,E2 -16777.245} C_VEL
LIN {X 0,Y 291.289,Z 314.2,A -85,B 0,C 180,E1 -16780.65,E2 -16780.65} C_VEL
LIN {X 0,Y 291.287,Z 314.2,A -85,B 0,C 180,E1 -16784.403,E2 -16784.403} C_VEL
LIN {X 0,Y 291.289,Z 314.201,A -85,B 0,C 180,E1 -16788.413,E2 -16788.413} C_VEL
LIN {X 0,Y 291.316,Z 314.196,A -85,B 0,C 180,E1 -16791.15,E2 -16791.15} C_VEL
LIN {X 0,Y 291.345,Z 314.195,A -85,B 0,C 180,E1 -16794.621,E2 -16794.621} C_VEL
LIN {X 0,Y 291.361,Z 314.19,A -85,B 0,C 180,E1 -16797.947,E2 -16797.947} C_VEL
LIN {X 0,Y 291.328,Z 314.197,A -85,B 0,C 180,E1 -16801.15,E2 -16801.15} C_VEL
LIN {X 0,Y 291.364,Z 314.191,A -85,B 0,C 180,E1 -16804.264,E2 -16804.264} C_VEL
LIN {X 0,Y 291.37,Z 314.193,A -85,B 0,C 180,E1 -16807.295,E2 -16807.295} C_VEL
LIN {X 0,Y 291.399,Z 314.185,A -85,B 0,C 180,E1 -16810.263,E2 -16810.263} C_VEL
LIN {X 0,Y 291.504,Z 314.172,A -85,B 0,C 180,E1 -16814.662,E2 -16814.662} C_VEL
LIN {X 0,Y 291.534,Z 314.168,A -85,B 0,C 180,E1 -16818.877,E2 -16818.877} C_VEL
LIN {X 0,Y 291.656,Z 314.154,A -85,B 0,C 180,E1 -16821.683,E2 -16821.683} C_VEL
LIN {X 0,Y 291.6,Z 314.16,A -85,B 0,C 180,E1 -16824.464,E2 -16824.464} C_VEL
LIN {X 0,Y 291.88,Z 314.124,A -85,B 0,C 180,E1 -16828.616,E2 -16828.616} C_VEL
LIN {X 0,Y 291.872,Z 314.128,A -85,B 0,C 180,E1 -16831.375,E2 -16831.375} C_VEL
LIN {X 0,Y 291.566,Z 314.269,A -85,B 0,C 180,E1 -16834.272,E2 -16834.272} C_VEL
LIN {X 0,Y 292.263,Z 317.299,A -85,B 0,C 180,E1 -16835.342,E2 -16835.342} C_VEL
LIN {X 0,Y 300.953,Z 340.539,A -85,B 0,C 180,E1 -16836.7,E2 -16836.7} C_VEL
LIN {X 0,Y 302.86,Z 346.704,A -85,B 0,C 180,E1 -16837.015,E2 -16837.015} C_VEL
LIN {X 0,Y 303.271,Z 350.577,A -85,B 0,C 180,E1 -16837.15,E2 -16837.15} C_VEL
LIN {X 0,Y 301.13,Z 424.64,A -85,B 0,C 180,E1 -16839.005,E2 -16839.005} C_VEL
LIN {X 0,Y 300.392,Z 438.225,A -85,B 0,C 180,E1 -16839.617,E2 -16839.617} C_VEL
LIN {X 0,Y 299.531,Z 449.978,A -85,B 0,C 180,E1 -16840.395,E2 -16840.395} C_VEL
LIN {X 0,Y 298.461,Z 461.097,A -85,B 0,C 180,E1 -16841.369,E2 -16841.369} C_VEL
LIN {X 0,Y 297.091,Z 472.169,A -85,B 0,C 180,E1 -16842.612,E2 -16842.612} C_VEL
LIN {X 0,Y 295.504,Z 483.826,A -85,B 0,C 180,E1 -16844.28,E2 -16844.28} C_VEL
LIN {X 0,Y 294.228,Z 493.043,A -85,B 0,C 180,E1 -16845.938,E2 -16845.938} C_VEL
LIN {X 0,Y 292.953,Z 501.297,A -85,B 0,C 180,E1 -16847.769,E2 -16847.769} C_VEL
LIN {X 0,Y 291.772,Z 509.5,A -85,B 0,C 180,E1 -16850.047,E2 -16850.047} C_VEL
LIN {X 0,Y 291.009,Z 515.005,A -85,B 0,C 180,E1 -16851.977,E2 -16851.977} C_VEL
LIN {X 0,Y 290.306,Z 520.201,A -85,B 0,C 180,E1 -16854.296,E2 -16854.296} C_VEL
LIN {X 0,Y 289.843,Z 523.442,A -85,B 0,C 180,E1 -16856.212,E2 -16856.212} C_VEL
LIN {X 0,Y 289.562,Z 525.09,A -85,B 0,C 180,E1 -16857.454,E2 -16857.454} C_VEL
LIN {X 0,Y 289.338,Z 526.674,A -85,B 0,C 180,E1 -16859.057,E2 -16859.057} C_VEL
LIN {X 0,Y 289.241,Z 528.169,A -85,B 0,C 180,E1 -16861.741,E2 -16861.741} C_VEL
LIN {X 0,Y 289.343,Z 528.166,A -85,B 0,C 180,E1 -16864.326,E2 -16864.326} C_VEL
LIN {X 0,Y 289.653,Z 526.874,A -85,B 0,C 180,E1 -16866.803,E2 -16866.803} C_VEL
LIN {X 0,Y 290.222,Z 524.393,A -85,B 0,C 180,E1 -16869.203,E2 -16869.203} C_VEL
LIN {X 0,Y 291.038,Z 520.747,A -85,B 0,C 180,E1 -16871.531,E2 -16871.531} C_VEL
LIN {X 0,Y 292.051,Z 515.924,A -85,B 0,C 180,E1 -16873.786,E2 -16873.786} C_VEL
LIN {X 0,Y 293.358,Z 509.743,A -85,B 0,C 180,E1 -16875.992,E2 -16875.992} C_VEL
LIN {X 0,Y 295.069,Z 501.95,A -85,B 0,C 180,E1 -16878.171,E2 -16878.171} C_VEL
LIN {X 0,Y 296.86,Z 493.341,A -85,B 0,C 180,E1 -16880.085,E2 -16880.085} C_VEL
LIN {X 0,Y 298.582,Z 483.951,A -85,B 0,C 180,E1 -16881.759,E2 -16881.759} C_VEL
LIN {X 0,Y 300.381,Z 473.546,A -85,B 0,C 180,E1 -16883.246,E2 -16883.246} C_VEL
LIN {X 0,Y 302.063,Z 462.423,A -85,B 0,C 180,E1 -16884.508,E2 -16884.508} C_VEL
LIN {X 0,Y 303.547,Z 450.345,A -85,B 0,C 180,E1 -16885.557,E2 -16885.557} C_VEL
LIN {X 0,Y 304.732,Z 437.27,A -85,B 0,C 180,E1 -16886.392,E2 -16886.392} C_VEL
LIN {X 0,Y 305.49,Z 425.274,A -85,B 0,C 180,E1 -16886.908,E2 -16886.908} C_VEL
LIN {X 0,Y 307.614,Z 365.414,A -85,B 0,C 180,E1 -16888.425,E2 -16888.425} C_VEL
LIN {X 0,Y 307.152,Z 361.638,A -85,B 0,C 180,E1 -16888.586,E2 -16888.586} C_VEL
LIN {X 0,Y 305.209,Z 357.094,A -85,B 0,C 180,E1 -16888.939,E2 -16888.939} C_VEL
LIN {X 0,Y 300.062,Z 348.479,A -85,B 0,C 180,E1 -16889.798,E2 -16889.798} C_VEL
LIN {X 0,Y 299.561,Z 347.296,A -85,B 0,C 180,E1 -16889.894,E2 -16889.894} C_VEL
LIN {X 0,Y 292.312,Z 331.669,A -85,B 0,C 180,E1 -16891.308,E2 -16891.308} C_VEL
LIN {X 0,Y 286.645,Z 321.118,A -85,B 0,C 180,E1 -16892.438,E2 -16892.438} C_VEL
LIN {X 0,Y 285.203,Z 318.232,A -85,B 0,C 180,E1 -16892.782,E2 -16892.782} C_VEL
LIN {X 0,Y 284.335,Z 315.076,A -85,B 0,C 180,E1 -16894.075,E2 -16894.075} C_VEL
LIN {X 0,Y 284.279,Z 315.08,A -85,B 0,C 180,E1 -16898.233,E2 -16898.233} C_VEL
LIN {X 0,Y 284.357,Z 315.064,A -85,B 0,C 180,E1 -16901.258,E2 -16901.258} C_VEL
LIN {X 0,Y 284.427,Z 315.056,A -85,B 0,C 180,E1 -16905.694,E2 -16905.694} C_VEL
LIN {X 0,Y 284.471,Z 315.045,A -85,B 0,C 180,E1 -16910.041,E2 -16910.041} C_VEL
LIN {X 0,Y 284.638,Z 315.023,A -85,B 0,C 180,E1 -16912.908,E2 -16912.908} C_VEL
LIN {X 0,Y 284.811,Z 315.005,A -85,B 0,C 180,E1 -16918.586,E2 -16918.586} C_VEL
LIN {X 0,Y 284.812,Z 315.007,A -85,B 0,C 180,E1 -16921.414,E2 -16921.414} C_VEL
LIN {X 0,Y 284.647,Z 315.02,A -85,B 0,C 180,E1 -16927.091,E2 -16927.091} C_VEL
LIN {X 0,Y 284.525,Z 315.043,A -85,B 0,C 180,E1 -16929.957,E2 -16929.957} C_VEL
LIN {X 0,Y 284.429,Z 315.054,A -85,B 0,C 180,E1 -16934.306,E2 -16934.306} C_VEL
LIN {X 0,Y 284.383,Z 315.059,A -85,B 0,C 180,E1 -16938.74,E2 -16938.74} C_VEL
LIN {X 0,Y 284.32,Z 315.063,A -85,B 0,C 180,E1 -16941.764,E2 -16941.764} C_VEL
LIN {X 0,Y 284.326,Z 315.055,A -85,B 0,C 180,E1 -16944.848,E2 -16944.848} C_VEL
LIN {X 0,Y 284.295,Z 315.061,A -85,B 0,C 180,E1 -16948.015,E2 -16948.015} C_VEL
LIN {X 0,Y 284.26,Z 315.071,A -85,B 0,C 180,E1 -16951.279,E2 -16951.279} C_VEL
LIN {X 0,Y 284.336,Z 315.061,A -85,B 0,C 180,E1 -16955.36,E2 -16955.36} C_VEL
LIN {X 0,Y 284.324,Z 315.064,A -85,B 0,C 180,E1 -16958.167,E2 -16958.167} C_VEL
LIN {X 0,Y 284.314,Z 315.072,A -85,B 0,C 180,E1 -16961.868,E2 -16961.868} C_VEL
LIN {X 0,Y 284.331,Z 315.072,A -85,B 0,C 180,E1 -16965.792,E2 -16965.792} C_VEL
LIN {X 0,Y 284.329,Z 315.069,A -85,B 0,C 180,E1 -16970.019,E2 -16970.019} C_VEL
LIN {X 0,Y 284.381,Z 315.208,A -85,B 0,C 180,E1 -16972.746,E2 -16972.746} C_VEL
LIN {X 0,Y 286.937,Z 324.951,A -85,B 0,C 180,E1 -16976.384,E2 -16976.384} C_VEL
LIN {X 0,Y 289.353,Z 335.321,A -85,B 0,C 180,E1 -16979.904,E2 -16979.904} C_VEL
LIN {X 0,Y 295.247,Z 348.726,A -85,B 0,C 180,E1 -16981.108,E2 -16981.108} C_VEL
LIN {X 0,Y 297.882,Z 362.249,A -85,B 0,C 180,E1 -16981.852,E2 -16981.852} C_VEL
LIN {X 0,Y 300.719,Z 381.763,A -85,B 0,C 180,E1 -16982.771,E2 -16982.771} C_VEL
LIN {X 0,Y 300.897,Z 385.847,A -85,B 0,C 180,E1 -16982.912,E2 -16982.912} C_VEL
LIN {X 0,Y 298.726,Z 444.736,A -85,B 0,C 180,E1 -16984.438,E2 -16984.438} C_VEL
LIN {X 0,Y 297.645,Z 458.322,A -85,B 0,C 180,E1 -16985.042,E2 -16985.042} C_VEL
LIN {X 0,Y 296.226,Z 470.68,A -85,B 0,C 180,E1 -16985.848,E2 -16985.848} C_VEL
LIN {X 0,Y 294.579,Z 481.825,A -85,B 0,C 180,E1 -16986.825,E2 -16986.825} C_VEL
LIN {X 0,Y 292.622,Z 493.438,A -85,B 0,C 180,E1 -16988.151,E2 -16988.151} C_VEL
LIN {X 0,Y 290.655,Z 503.936,A -85,B 0,C 180,E1 -16989.667,E2 -16989.667} C_VEL
LIN {X 0,Y 288.943,Z 512.549,A -85,B 0,C 180,E1 -16991.205,E2 -16991.205} C_VEL
LIN {X 0,Y 287.007,Z 521.927,A -85,B 0,C 180,E1 -16993.284,E2 -16993.284} C_VEL
LIN {X 0,Y 285.425,Z 529.468,A -85,B 0,C 180,E1 -16995.387,E2 -16995.387} C_VEL
LIN {X 0,Y 283.963,Z 536.464,A -85,B 0,C 180,E1 -16997.861,E2 -16997.861} C_VEL
LIN {X 0,Y 283.162,Z 541.102,A -85,B 0,C 180,E1 -17000,E2 -17000} C_VEL
LIN {X 0,Y 282.672,Z 544.652,A -85,B 0,C 180,E1 -17002.146,E2 -17002.146} C_VEL
LIN {X 0,Y 282.368,Z 547.493,A -85,B 0,C 180,E1 -17004.613,E2 -17004.613} C_VEL
LIN {X 0,Y 282.377,Z 549.126,A -85,B 0,C 180,E1 -17007.152,E2 -17007.152} C_VEL
LIN {X 0,Y 282.371,Z 549.486,A -85,B 0,C 180,E1 -17008.579,E2 -17008.579} C_VEL
LIN {X 0,Y 282.412,Z 549.454,A -85,B 0,C 180,E1 -17010.005,E2 -17010.005} C_VEL
LIN {X 0,Y 282.382,Z 548.989,A -85,B 0,C 180,E1 -17011.431,E2 -17011.431} C_VEL
LIN {X 0,Y 282.409,Z 548.099,A -85,B 0,C 180,E1 -17012.857,E2 -17012.857} C_VEL
LIN {X 0,Y 282.381,Z 545.464,A -85,B 0,C 180,E1 -17015.415,E2 -17015.415} C_VEL
LIN {X 0,Y 282.668,Z 541.61,A -85,B 0,C 180,E1 -17017.864,E2 -17017.864} C_VEL
LIN {X 0,Y 283.092,Z 537.019,A -85,B 0,C 180,E1 -17020.012,E2 -17020.012} C_VEL
LIN {X 0,Y 283.934,Z 530.028,A -85,B 0,C 180,E1 -17022.512,E2 -17022.512} C_VEL
LIN {X 0,Y 285.123,Z 522.45,A -85,B 0,C 180,E1 -17024.638,E2 -17024.638} C_VEL
LIN {X 0,Y 286.483,Z 513.725,A -85,B 0,C 180,E1 -17026.598,E2 -17026.598} C_VEL
LIN {X 0,Y 287.778,Z 504.161,A -85,B 0,C 180,E1 -17028.33,E2 -17028.33} C_VEL
LIN {X 0,Y 289.353,Z 493.439,A -85,B 0,C 180,E1 -17029.883,E2 -17029.883} C_VEL
LIN {X 0,Y 290.755,Z 483.094,A -85,B 0,C 180,E1 -17031.076,E2 -17031.076} C_VEL
LIN {X 0,Y 292.178,Z 470.768,A -85,B 0,C 180,E1 -17032.173,E2 -17032.173} C_VEL
LIN {X 0,Y 293.424,Z 457.14,A -85,B 0,C 180,E1 -17033.049,E2 -17033.049} C_VEL
LIN {X 0,Y 294.226,Z 444.292,A -85,B 0,C 180,E1 -17033.587,E2 -17033.587} C_VEL
LIN {X 0,Y 295.98,Z 383.114,A -85,B 0,C 180,E1 -17035.153,E2 -17035.153} C_VEL
LIN {X 0,Y 291.837,Z 352.883,A -85,B 0,C 180,E1 -17036.323,E2 -17036.323} C_VEL
LIN {X 0,Y 289.369,Z 338.699,A -85,B 0,C 180,E1 -17036.929,E2 -17036.929} C_VEL
LIN {X 0,Y 289.003,Z 337.199,A -85,B 0,C 180,E1 -17037.033,E2 -17037.033} C_VEL
LIN {X 0,Y 287.034,Z 327.449,A -85,B 0,C 180,E1 -17040.131,E2 -17040.131} C_VEL
LIN {X 0,Y 284.687,Z 316.594,A -85,B 0,C 180,E1 -17043.744,E2 -17043.744} C_VEL
LIN {X 0,Y 284.332,Z 315.068,A -85,B 0,C 180,E1 -17044.326,E2 -17044.326} C_VEL
LIN {X 0,Y 284.318,Z 315.072,A -85,B 0,C 180,E1 -17048.171,E2 -17048.171} C_VEL
LIN {X 0,Y 284.276,Z 315.077,A -85,B 0,C 180,E1 -17052.126,E2 -17052.126} C_VEL
LIN {X 0,Y 284.262,Z 315.079,A -85,B 0,C 180,E1 -17056.19,E2 -17056.19} C_VEL
LIN {X 0,Y 284.313,Z 315.068,A -85,B 0,C 180,E1 -17060.025,E2 -17060.025} C_VEL
LIN {X 0,Y 284.327,Z 315.066,A -85,B 0,C 180,E1 -17063.613,E2 -17063.613} C_VEL
LIN {X 0,Y 284.311,Z 315.07,A -85,B 0,C 180,E1 -17067.191,E2 -17067.191} C_VEL
LIN {X 0,Y 284.354,Z 315.062,A -85,B 0,C 180,E1 -17070.375,E2 -17070.375} C_VEL
LIN {X 0,Y 284.378,Z 315.059,A -85,B 0,C 180,E1 -17073.587,E2 -17073.587} C_VEL
LIN {X 0,Y 284.335,Z 315.067,A -85,B 0,C 180,E1 -17076.704,E2 -17076.704} C_VEL
LIN {X 0,Y 284.334,Z 315.061,A -85,B 0,C 180,E1 -17081.257,E2 -17081.257} C_VEL
LIN {X 0,Y 284.464,Z 315.044,A -85,B 0,C 180,E1 -17085.696,E2 -17085.696} C_VEL
LIN {X 0,Y 284.516,Z 315.042,A -85,B 0,C 180,E1 -17090.043,E2 -17090.043} C_VEL
LIN {X 0,Y 284.682,Z 315.021,A -85,B 0,C 180,E1 -17092.91,E2 -17092.91} C_VEL
LIN {X 0,Y 284.852,Z 314.985,A -85,B 0,C 180,E1 -17098.586,E2 -17098.586} C_VEL
LIN {X 0,Y 284.851,Z 314.996,A -85,B 0,C 180,E1 -17101.414,E2 -17101.414} C_VEL
LIN {X 0,Y 284.592,Z 315.032,A -85,B 0,C 180,E1 -17106.558,E2 -17106.558} C_VEL
LIN {X 0,Y 284.513,Z 315.041,A -85,B 0,C 180,E1 -17109.957,E2 -17109.957} C_VEL
LIN {X 0,Y 284.464,Z 315.049,A -85,B 0,C 180,E1 -17114.304,E2 -17114.304} C_VEL
LIN {X 0,Y 284.332,Z 315.059,A -85,B 0,C 180,E1 -17118.743,E2 -17118.743} C_VEL
LIN {X 0,Y 284.312,Z 315.067,A -85,B 0,C 180,E1 -17123.298,E2 -17123.298} C_VEL
LIN {X 0,Y 284.286,Z 315.066,A -85,B 0,C 180,E1 -17127.128,E2 -17127.128} C_VEL
LIN {X 0,Y 284.275,Z 315.061,A -85,B 0,C 180,E1 -17130.082,E2 -17130.082} C_VEL
LIN {X 0,Y 284.289,Z 315.06,A -85,B 0,C 180,E1 -17132.948,E2 -17132.948} C_VEL
LIN {X 0,Y 284.32,Z 315.068,A -85,B 0,C 180,E1 -17136.388,E2 -17136.388} C_VEL
LIN {X 0,Y 284.259,Z 315.075,A -85,B 0,C 180,E1 -17140.003,E2 -17140.003} C_VEL
LIN {X 0,Y 284.238,Z 315.076,A -85,B 0,C 180,E1 -17144.186,E2 -17144.186} C_VEL
LIN {X 0,Y 284.236,Z 315.077,A -85,B 0,C 180,E1 -17148.115,E2 -17148.115} C_VEL
LIN {X 0,Y 284.279,Z 315.073,A -85,B 0,C 180,E1 -17152.29,E2 -17152.29} C_VEL
LIN {X 0,Y 284.297,Z 315.069,A -85,B 0,C 180,E1 -17155.346,E2 -17155.346} C_VEL
LIN {X 0,Y 284.278,Z 315.076,A -85,B 0,C 180,E1 -17158.721,E2 -17158.721} C_VEL
LIN {X 0,Y 284.334,Z 315.069,A -85,B 0,C 180,E1 -17162.852,E2 -17162.852} C_VEL
LIN {X 0,Y 284.334,Z 315.066,A -85,B 0,C 180,E1 -17166.701,E2 -17166.701} C_VEL
LIN {X 0,Y 284.34,Z 315.069,A -85,B 0,C 180,E1 -17171.254,E2 -17171.254} C_VEL
LIN {X 0,Y 284.469,Z 315.05,A -85,B 0,C 180,E1 -17175.693,E2 -17175.693} C_VEL
LIN {X 0,Y 284.519,Z 315.042,A -85,B 0,C 180,E1 -17180.039,E2 -17180.039} C_VEL
LIN {X 0,Y 284.645,Z 315.026,A -85,B 0,C 180,E1 -17182.905,E2 -17182.905} C_VEL
LIN {X 0,Y 284.847,Z 315,A -85,B 0,C 180,E1 -17188.582,E2 -17188.582} C_VEL
LIN {X 0,Y 284.839,Z 315.004,A -85,B 0,C 180,E1 -17191.409,E2 -17191.409} C_VEL
LIN {X 0,Y 284.545,Z 315.144,A -85,B 0,C 180,E1 -17193.845,E2 -17193.845} C_VEL
LIN {X 0,Y 285.024,Z 317.587,A -85,B 0,C 180,E1 -17194.724,E2 -17194.724} C_VEL
LIN {X 0,Y 292.509,Z 336.836,A -85,B 0,C 180,E1 -17195.917,E2 -17195.917} C_VEL
LIN {X 0,Y 296.377,Z 348.258,A -85,B 0,C 180,E1 -17196.548,E2 -17196.548} C_VEL
LIN {X 0,Y 296.662,Z 351.866,A -85,B 0,C 180,E1 -17196.67,E2 -17196.67} C_VEL
LIN {X 0,Y 294.476,Z 424.622,A -85,B 0,C 180,E1 -17198.53,E2 -17198.53} C_VEL
LIN {X 0,Y 293.713,Z 438.365,A -85,B 0,C 180,E1 -17199.159,E2 -17199.159} C_VEL
LIN {X 0,Y 292.787,Z 450.647,A -85,B 0,C 180,E1 -17199.992,E2 -17199.992} C_VEL
LIN {X 0,Y 291.482,Z 462.902,A -85,B 0,C 180,E1 -17201.116,E2 -17201.116} C_VEL
LIN {X 0,Y 290.118,Z 473.813,A -85,B 0,C 180,E1 -17202.41,E2 -17202.41} C_VEL
LIN {X 0,Y 288.69,Z 483.808,A -85,B 0,C 180,E1 -17203.886,E2 -17203.886} C_VEL
LIN {X 0,Y 287.326,Z 493.192,A -85,B 0,C 180,E1 -17205.603,E2 -17205.603} C_VEL
LIN {X 0,Y 285.992,Z 501.612,A -85,B 0,C 180,E1 -17207.514,E2 -17207.514} C_VEL
LIN {X 0,Y 284.761,Z 509.724,A -85,B 0,C 180,E1 -17209.82,E2 -17209.82} C_VEL
LIN {X 0,Y 283.98,Z 515.208,A -85,B 0,C 180,E1 -17211.785,E2 -17211.785} C_VEL
LIN {X 0,Y 283.262,Z 520.418,A -85,B 0,C 180,E1 -17214.158,E2 -17214.158} C_VEL
LIN {X 0,Y 282.658,Z 524.291,A -85,B 0,C 180,E1 -17216.58,E2 -17216.58} C_VEL
LIN {X 0,Y 282.219,Z 527.178,A -85,B 0,C 180,E1 -17219.355,E2 -17219.355} C_VEL
LIN {X 0,Y 282.128,Z 528.497,A -85,B 0,C 180,E1 -17222.117,E2 -17222.117} C_VEL
LIN {X 0,Y 282.28,Z 528.345,A -85,B 0,C 180,E1 -17224.753,E2 -17224.753} C_VEL
LIN {X 0,Y 282.646,Z 526.937,A -85,B 0,C 180,E1 -17227.28,E2 -17227.28} C_VEL
LIN {X 0,Y 283.306,Z 524.34,A -85,B 0,C 180,E1 -17229.734,E2 -17229.734} C_VEL
LIN {X 0,Y 284.173,Z 520.579,A -85,B 0,C 180,E1 -17232.103,E2 -17232.103} C_VEL
LIN {X 0,Y 285.309,Z 515.581,A -85,B 0,C 180,E1 -17234.409,E2 -17234.409} C_VEL
LIN {X 0,Y 286.736,Z 509.254,A -85,B 0,C 180,E1 -17236.663,E2 -17236.663} C_VEL
LIN {X 0,Y 288.592,Z 501.277,A -85,B 0,C 180,E1 -17238.889,E2 -17238.889} C_VEL
LIN {X 0,Y 290.357,Z 492.855,A -85,B 0,C 180,E1 -17240.752,E2 -17240.752} C_VEL
LIN {X 0,Y 292.25,Z 482.998,A -85,B 0,C 180,E1 -17242.509,E2 -17242.509} C_VEL
LIN {X 0,Y 294.295,Z 472.067,A -85,B 0,C 180,E1 -17244.049,E2 -17244.049} C_VEL
LIN {X 0,Y 296.045,Z 459.975,A -85,B 0,C 180,E1 -17245.382,E2 -17245.382} C_VEL
LIN {X 0,Y 297.511,Z 448.252,A -85,B 0,C 180,E1 -17246.363,E2 -17246.363} C_VEL
LIN {X 0,Y 298.58,Z 436.041,A -85,B 0,C 180,E1 -17247.123,E2 -17247.123} C_VEL
LIN {X 0,Y 299.439,Z 422.616,A -85,B 0,C 180,E1 -17247.651,E2 -17247.651} C_VEL
LIN {X 0,Y 301.966,Z 353.444,A -85,B 0,C 180,E1 -17249.423,E2 -17249.423} C_VEL
LIN {X 0,Y 299.561,Z 347.296,A -85,B 0,C 180,E1 -17249.894,E2 -17249.894} C_VEL
LIN {X 0,Y 296.987,Z 342.589,A -85,B 0,C 180,E1 -17250.357,E2 -17250.357} C_VEL
LIN {X 0,Y 293.622,Z 338.628,A -85,B 0,C 180,E1 -17250.913,E2 -17250.913} C_VEL
LIN {X 0,Y 286.24,Z 331.487,A -85,B 0,C 180,E1 -17252.152,E2 -17252.152} C_VEL
LIN {X 0,Y 282.987,Z 327.449,A -85,B 0,C 180,E1 -17252.759,E2 -17252.759} C_VEL
LIN {X 0,Y 282.072,Z 325.936,A -85,B 0,C 180,E1 -17252.948,E2 -17252.948} C_VEL
LIN {X 0,Y 278.046,Z 318.656,A -85,B 0,C 180,E1 -17253.848,E2 -17253.848} C_VEL
LIN {X 0,Y 277.26,Z 315.955,A -85,B 0,C 180,E1 -17255.001,E2 -17255.001} C_VEL
LIN {X 0,Y 277.306,Z 315.948,A -85,B 0,C 180,E1 -17259.648,E2 -17259.648} C_VEL
LIN {X 0,Y 277.377,Z 315.932,A -85,B 0,C 180,E1 -17264.295,E2 -17264.295} C_VEL
LIN {X 0,Y 277.387,Z 315.933,A -85,B 0,C 180,E1 -17268.305,E2 -17268.305} C_VEL
LIN {X 0,Y 277.557,Z 315.911,A -85,B 0,C 180,E1 -17271.261,E2 -17271.261} C_VEL
LIN {X 0,Y 277.522,Z 315.915,A -85,B 0,C 180,E1 -17274.186,E2 -17274.186} C_VEL
LIN {X 0,Y 277.777,Z 315.881,A -85,B 0,C 180,E1 -17278.55,E2 -17278.55} C_VEL
LIN {X 0,Y 277.778,Z 315.883,A -85,B 0,C 180,E1 -17281.45,E2 -17281.45} C_VEL
LIN {X 0,Y 277.603,Z 315.896,A -85,B 0,C 180,E1 -17287.272,E2 -17287.272} C_VEL
LIN {X 0,Y 277.465,Z 315.923,A -85,B 0,C 180,E1 -17290.213,E2 -17290.213} C_VEL
LIN {X 0,Y 277.375,Z 315.934,A -85,B 0,C 180,E1 -17294.677,E2 -17294.677} C_VEL
LIN {X 0,Y 277.332,Z 315.932,A -85,B 0,C 180,E1 -17299.235,E2 -17299.235} C_VEL
LIN {X 0,Y 277.308,Z 315.93,A -85,B 0,C 180,E1 -17303.922,E2 -17303.922} C_VEL
LIN {X 0,Y 277.29,Z 315.936,A -85,B 0,C 180,E1 -17307.508,E2 -17307.508} C_VEL
LIN {X 0,Y 277.239,Z 315.949,A -85,B 0,C 180,E1 -17310.486,E2 -17310.486} C_VEL
LIN {X 0,Y 277.223,Z 315.952,A -85,B 0,C 180,E1 -17313.899,E2 -17313.899} C_VEL
LIN {X 0,Y 277.276,Z 315.945,A -85,B 0,C 180,E1 -17317.468,E2 -17317.468} C_VEL
LIN {X 0,Y 277.268,Z 315.946,A -85,B 0,C 180,E1 -17321.226,E2 -17321.226} C_VEL
LIN {X 0,Y 277.262,Z 315.956,A -85,B 0,C 180,E1 -17325.214,E2 -17325.214} C_VEL
LIN {X 0,Y 277.273,Z 315.951,A -85,B 0,C 180,E1 -17329.5,E2 -17329.5} C_VEL
LIN {X 0,Y 277.284,Z 316.036,A -85,B 0,C 180,E1 -17331.788,E2 -17331.788} C_VEL
LIN {X 0,Y 279.576,Z 324.3,A -85,B 0,C 180,E1 -17335.056,E2 -17335.056} C_VEL
LIN {X 0,Y 281.77,Z 333.553,A -85,B 0,C 180,E1 -17338.421,E2 -17338.421} C_VEL
LIN {X 0,Y 282.051,Z 334.891,A -85,B 0,C 180,E1 -17338.848,E2 -17338.848} C_VEL
LIN {X 0,Y 288.24,Z 348.274,A -85,B 0,C 180,E1 -17340.171,E2 -17340.171} C_VEL
LIN {X 0,Y 289.917,Z 352.698,A -85,B 0,C 180,E1 -17340.539,E2 -17340.539} C_VEL
LIN {X 0,Y 293.46,Z 373.406,A -85,B 0,C 180,E1 -17341.652,E2 -17341.652} C_VEL
LIN {X 0,Y 294.895,Z 384.7,A -85,B 0,C 180,E1 -17342.173,E2 -17342.173} C_VEL
LIN {X 0,Y 292.511,Z 445.325,A -85,B 0,C 180,E1 -17343.781,E2 -17343.781} C_VEL
LIN {X 0,Y 291.344,Z 459.012,A -85,B 0,C 180,E1 -17344.416,E2 -17344.416} C_VEL
LIN {X 0,Y 289.802,Z 471.599,A -85,B 0,C 180,E1 -17345.278,E2 -17345.278} C_VEL
LIN {X 0,Y 288.103,Z 482.452,A -85,B 0,C 180,E1 -17346.272,E2 -17346.272} C_VEL
LIN {X 0,Y 286.079,Z 493.881,A -85,B 0,C 180,E1 -17347.624,E2 -17347.624} C_VEL
LIN {X 0,Y 284.023,Z 504.235,A -85,B 0,C 180,E1 -17349.17,E2 -17349.17} C_VEL
LIN {X 0,Y 282.224,Z 512.734,A -85,B 0,C 180,E1 -17350.74,E2 -17350.74} C_VEL
LIN {X 0,Y 280.216,Z 521.991,A -85,B 0,C 180,E1 -17352.867,E2 -17352.867} C_VEL
LIN {X 0,Y 278.549,Z 529.476,A -85,B 0,C 180,E1 -17355.018,E2 -17355.018} C_VEL
LIN {X 0,Y 276.979,Z 536.401,A -85,B 0,C 180,E1 -17357.55,E2 -17357.55} C_VEL
LIN {X 0,Y 276.153,Z 540.993,A -85,B 0,C 180,E1 -17359.744,E2 -17359.744} C_VEL
LIN {X 0,Y 275.601,Z 544.505,A -85,B 0,C 180,E1 -17361.943,E2 -17361.943} C_VEL
LIN {X 0,Y 275.282,Z 547.456,A -85,B 0,C 180,E1 -17364.673,E2 -17364.673} C_VEL
LIN {X 0,Y 275.283,Z 548.888,A -85,B 0,C 180,E1 -17367.078,E2 -17367.078} C_VEL
LIN {X 0,Y 275.294,Z 549.229,A -85,B 0,C 180,E1 -17368.542,E2 -17368.542} C_VEL
LIN {X 0,Y 275.331,Z 549.176,A -85,B 0,C 180,E1 -17370.005,E2 -17370.005} C_VEL
LIN {X 0,Y 275.305,Z 548.677,A -85,B 0,C 180,E1 -17371.467,E2 -17371.467} C_VEL
LIN {X 0,Y 275.314,Z 547.767,A -85,B 0,C 180,E1 -17372.931,E2 -17372.931} C_VEL
LIN {X 0,Y 275.296,Z 545.335,A -85,B 0,C 180,E1 -17375.358,E2 -17375.358} C_VEL
LIN {X 0,Y 275.592,Z 541.189,A -85,B 0,C 180,E1 -17378.067,E2 -17378.067} C_VEL
LIN {X 0,Y 276.063,Z 536.546,A -85,B 0,C 180,E1 -17380.269,E2 -17380.269} C_VEL
LIN {X 0,Y 276.97,Z 529.491,A -85,B 0,C 180,E1 -17382.832,E2 -17382.832} C_VEL
LIN {X 0,Y 278.179,Z 521.847,A -85,B 0,C 180,E1 -17385.012,E2 -17385.012} C_VEL
LIN {X 0,Y 279.389,Z 514.654,A -85,B 0,C 180,E1 -17386.677,E2 -17386.677} C_VEL
LIN {X 0,Y 280.83,Z 504.433,A -85,B 0,C 180,E1 -17388.611,E2 -17388.611} C_VEL
LIN {X 0,Y 282.452,Z 493.817,A -85,B 0,C 180,E1 -17390.2,E2 -17390.2} C_VEL
LIN {X 0,Y 284.117,Z 481.993,A -85,B 0,C 180,E1 -17391.593,E2 -17391.593} C_VEL
LIN {X 0,Y 285.624,Z 469.366,A -85,B 0,C 180,E1 -17392.709,E2 -17392.709} C_VEL
LIN {X 0,Y 286.801,Z 456.081,A -85,B 0,C 180,E1 -17393.565,E2 -17393.565} C_VEL
LIN {X 0,Y 287.634,Z 442.544,A -85,B 0,C 180,E1 -17394.114,E2 -17394.114} C_VEL
LIN {X 0,Y 289.285,Z 382.649,A -85,B 0,C 180,E1 -17395.686,E2 -17395.686} C_VEL
LIN {X 0,Y 285.113,Z 352.787,A -85,B 0,C 180,E1 -17396.88,E2 -17396.88} C_VEL
LIN {X 0,Y 282.986,Z 340.636,A -85,B 0,C 180,E1 -17397.418,E2 -17397.418} C_VEL
LIN {X 0,Y 281.785,Z 336.943,A -85,B 0,C 180,E1 -17397.661,E2 -17397.661} C_VEL
LIN {X 0,Y 279.114,Z 324.042,A -85,B 0,C 180,E1 -17401.926,E2 -17401.926} C_VEL
LIN {X 0,Y 277.286,Z 315.945,A -85,B 0,C 180,E1 -17404.773,E2 -17404.773} C_VEL
LIN {X 0,Y 277.271,Z 315.949,A -85,B 0,C 180,E1 -17408.209,E2 -17408.209} C_VEL
LIN {X 0,Y 277.222,Z 315.953,A -85,B 0,C 180,E1 -17412.676,E2 -17412.676} C_VEL
LIN {X 0,Y 277.216,Z 315.955,A -85,B 0,C 180,E1 -17416.803,E2 -17416.803} C_VEL
LIN {X 0,Y 277.238,Z 315.953,A -85,B 0,C 180,E1 -17420.672,E2 -17420.672} C_VEL
LIN {X 0,Y 277.283,Z 315.946,A -85,B 0,C 180,E1 -17424.341,E2 -17424.341} C_VEL
LIN {X 0,Y 277.246,Z 315.949,A -85,B 0,C 180,E1 -17427.836,E2 -17427.836} C_VEL
LIN {X 0,Y 277.268,Z 315.947,A -85,B 0,C 180,E1 -17431.21,E2 -17431.21} C_VEL
LIN {X 0,Y 277.311,Z 315.941,A -85,B 0,C 180,E1 -17434.479,E2 -17434.479} C_VEL
LIN {X 0,Y 277.265,Z 315.945,A -85,B 0,C 180,E1 -17437.653,E2 -17437.653} C_VEL
LIN {X 0,Y 277.287,Z 315.943,A -85,B 0,C 180,E1 -17440.762,E2 -17440.762} C_VEL
LIN {X 0,Y 277.411,Z 315.922,A -85,B 0,C 180,E1 -17445.325,E2 -17445.325} C_VEL
LIN {X 0,Y 277.457,Z 315.922,A -85,B 0,C 180,E1 -17449.787,E2 -17449.787} C_VEL
LIN {X 0,Y 277.637,Z 315.898,A -85,B 0,C 180,E1 -17452.729,E2 -17452.729} C_VEL
LIN {X 0,Y 277.819,Z 315.859,A -85,B 0,C 180,E1 -17458.55,E2 -17458.55} C_VEL
LIN {X 0,Y 277.818,Z 315.872,A -85,B 0,C 180,E1 -17461.45,E2 -17461.45} C_VEL
LIN {X 0,Y 277.593,Z 315.906,A -85,B 0,C 180,E1 -17467.273,E2 -17467.273} C_VEL
LIN {X 0,Y 277.455,Z 315.918,A -85,B 0,C 180,E1 -17470.213,E2 -17470.213} C_VEL
LIN {X 0,Y 277.411,Z 315.927,A -85,B 0,C 180,E1 -17474.675,E2 -17474.675} C_VEL
LIN {X 0,Y 277.286,Z 315.937,A -85,B 0,C 180,E1 -17479.238,E2 -17479.238} C_VEL
LIN {X 0,Y 277.261,Z 315.949,A -85,B 0,C 180,E1 -17483.927,E2 -17483.927} C_VEL
LIN {X 0,Y 277.236,Z 315.944,A -85,B 0,C 180,E1 -17487.467,E2 -17487.467} C_VEL
LIN {X 0,Y 277.233,Z 315.932,A -85,B 0,C 180,E1 -17490.465,E2 -17490.465} C_VEL
LIN {X 0,Y 277.244,Z 315.938,A -85,B 0,C 180,E1 -17493.896,E2 -17493.896} C_VEL
LIN {X 0,Y 277.235,Z 315.948,A -85,B 0,C 180,E1 -17497.475,E2 -17497.475} C_VEL
LIN {X 0,Y 277.176,Z 315.954,A -85,B 0,C 180,E1 -17501.243,E2 -17501.243} C_VEL
LIN {X 0,Y 277.179,Z 315.956,A -85,B 0,C 180,E1 -17505.231,E2 -17505.231} C_VEL
LIN {X 0,Y 277.18,Z 315.953,A -85,B 0,C 180,E1 -17509.523,E2 -17509.523} C_VEL
LIN {X 0,Y 277.229,Z 315.953,A -85,B 0,C 180,E1 -17512.522,E2 -17512.522} C_VEL
LIN {X 0,Y 277.236,Z 315.947,A -85,B 0,C 180,E1 -17516.1,E2 -17516.1} C_VEL
LIN {X 0,Y 277.235,Z 315.95,A -85,B 0,C 180,E1 -17519.532,E2 -17519.532} C_VEL
LIN {X 0,Y 277.296,Z 315.946,A -85,B 0,C 180,E1 -17522.854,E2 -17522.854} C_VEL
LIN {X 0,Y 277.288,Z 315.942,A -85,B 0,C 180,E1 -17526.072,E2 -17526.072} C_VEL
LIN {X 0,Y 277.292,Z 315.944,A -85,B 0,C 180,E1 -17530.759,E2 -17530.759} C_VEL
LIN {X 0,Y 277.415,Z 315.931,A -85,B 0,C 180,E1 -17535.321,E2 -17535.321} C_VEL
LIN {X 0,Y 277.462,Z 315.922,A -85,B 0,C 180,E1 -17539.783,E2 -17539.783} C_VEL
LIN {X 0,Y 277.604,Z 315.903,A -85,B 0,C 180,E1 -17542.724,E2 -17542.724} C_VEL
LIN {X 0,Y 277.813,Z 315.877,A -85,B 0,C 180,E1 -17548.546,E2 -17548.546} C_VEL
LIN {X 0,Y 277.806,Z 315.88,A -85,B 0,C 180,E1 -17551.445,E2 -17551.445} C_VEL
LIN {X 0,Y 277.594,Z 316.11,A -85,B 0,C 180,E1 -17553.442,E2 -17553.442} C_VEL
LIN {X 0,Y 277.845,Z 317.847,A -85,B 0,C 180,E1 -17554.075,E2 -17554.075} C_VEL
LIN {X 0,Y 285.778,Z 337.931,A -85,B 0,C 180,E1 -17555.384,E2 -17555.384} C_VEL
LIN {X 0,Y 290.01,Z 350.496,A -85,B 0,C 180,E1 -17556.099,E2 -17556.099} C_VEL
LIN {X 0,Y 287.942,Z 420.969,A -85,B 0,C 180,E1 -17557.93,E2 -17557.93} C_VEL
LIN {X 0,Y 287.255,Z 434.778,A -85,B 0,C 180,E1 -17558.48,E2 -17558.48} C_VEL
LIN {X 0,Y 286.324,Z 447.289,A -85,B 0,C 180,E1 -17559.264,E2 -17559.264} C_VEL
LIN {X 0,Y 285.256,Z 459.078,A -85,B 0,C 180,E1 -17560.283,E2 -17560.283} C_VEL
LIN {X 0,Y 283.705,Z 470.982,A -85,B 0,C 180,E1 -17561.606,E2 -17561.606} C_VEL
LIN {X 0,Y 282.117,Z 482.137,A -85,B 0,C 180,E1 -17563.21,E2 -17563.21} C_VEL
LIN {X 0,Y 280.737,Z 491.346,A -85,B 0,C 180,E1 -17564.863,E2 -17564.863} C_VEL
LIN {X 0,Y 279.541,Z 498.846,A -85,B 0,C 180,E1 -17566.493,E2 -17566.493} C_VEL
LIN {X 0,Y 278.171,Z 507.421,A -85,B 0,C 180,E1 -17568.785,E2 -17568.785} C_VEL
LIN {X 0,Y 277.092,Z 514.379,A -85,B 0,C 180,E1 -17571.181,E2 -17571.181} C_VEL
LIN {X 0,Y 276.283,Z 519.98,A -85,B 0,C 180,E1 -17573.686,E2 -17573.686} C_VEL
LIN {X 0,Y 275.774,Z 523.344,A -85,B 0,C 180,E1 -17575.666,E2 -17575.666} C_VEL
LIN {X 0,Y 275.403,Z 525.557,A -85,B 0,C 180,E1 -17577.337,E2 -17577.337} C_VEL
LIN {X 0,Y 275.098,Z 527.687,A -85,B 0,C 180,E1 -17579.703,E2 -17579.703} C_VEL
LIN {X 0,Y 275.049,Z 528.806,A -85,B 0,C 180,E1 -17582.519,E2 -17582.519} C_VEL
LIN {X 0,Y 275.228,Z 528.53,A -85,B 0,C 180,E1 -17585.201,E2 -17585.201} C_VEL
LIN {X 0,Y 275.696,Z 526.995,A -85,B 0,C 180,E1 -17587.791,E2 -17587.791} C_VEL
LIN {X 0,Y 276.408,Z 524.258,A -85,B 0,C 180,E1 -17590.289,E2 -17590.289} C_VEL
LIN {X 0,Y 277.36,Z 520.358,A -85,B 0,C 180,E1 -17592.707,E2 -17592.707} C_VEL
LIN {X 0,Y 278.581,Z 515.248,A -85,B 0,C 180,E1 -17595.059,E2 -17595.059} C_VEL
LIN {X 0,Y 280.163,Z 508.76,A -85,B 0,C 180,E1 -17597.366,E2 -17597.366} C_VEL
LIN {X 0,Y 281.913,Z 501.66,A -85,B 0,C 180,E1 -17599.368,E2 -17599.368} C_VEL
LIN {X 0,Y 283.759,Z 493.324,A -85,B 0,C 180,E1 -17601.264,E2 -17601.264} C_VEL
LIN {X 0,Y 285.732,Z 483.531,A -85,B 0,C 180,E1 -17603.059,E2 -17603.059} C_VEL
LIN {X 0,Y 287.656,Z 473.672,A -85,B 0,C 180,E1 -17604.497,E2 -17604.497} C_VEL
LIN {X 0,Y 289.5,Z 462.281,A -85,B 0,C 180,E1 -17605.825,E2 -17605.825} C_VEL
LIN {X 0,Y 291.198,Z 449.336,A -85,B 0,C 180,E1 -17606.963,E2 -17606.963} C_VEL
LIN {X 0,Y 292.397,Z 436.493,A -85,B 0,C 180,E1 -17607.788,E2 -17607.788} C_VEL
LIN {X 0,Y 293.292,Z 423.516,A -85,B 0,C 180,E1 -17608.315,E2 -17608.315} C_VEL
LIN {X 0,Y 295.799,Z 355.087,A -85,B 0,C 180,E1 -17610.119,E2 -17610.119} C_VEL
LIN {X 0,Y 290.657,Z 342.87,A -85,B 0,C 180,E1 -17611.172,E2 -17611.172} C_VEL
LIN {X 0,Y 284.176,Z 329.777,A -85,B 0,C 180,E1 -17612.506,E2 -17612.506} C_VEL
LIN {X 0,Y 282.072,Z 325.936,A -85,B 0,C 180,E1 -17612.948,E2 -17612.948} C_VEL
LIN {X 0,Y 279.904,Z 322.936,A -85,B 0,C 180,E1 -17613.386,E2 -17613.386} C_VEL
LIN {X 0,Y 276.291,Z 319.913,A -85,B 0,C 180,E1 -17614.061,E2 -17614.061} C_VEL
LIN {X 0,Y 273.977,Z 318.813,A -85,B 0,C 180,E1 -17614.524,E2 -17614.524} C_VEL
LIN {X 0,Y 271.244,Z 318.07,A -85,B 0,C 180,E1 -17615.303,E2 -17615.303} C_VEL
LIN {X 0,Y 270.237,Z 316.859,A -85,B 0,C 180,E1 -17616.027,E2 -17616.027} C_VEL
LIN {X 0,Y 270.226,Z 316.833,A -85,B 0,C 180,E1 -17616.099,E2 -17616.099} C_VEL
LIN {X 0,Y 270.261,Z 316.827,A -85,B 0,C 180,E1 -17620.241,E2 -17620.241} C_VEL
LIN {X 0,Y 270.342,Z 316.813,A -85,B 0,C 180,E1 -17624.932,E2 -17624.932} C_VEL
LIN {X 0,Y 270.368,Z 316.8,A -85,B 0,C 180,E1 -17629.516,E2 -17629.516} C_VEL
LIN {X 0,Y 270.552,Z 316.777,A -85,B 0,C 180,E1 -17632.537,E2 -17632.537} C_VEL
LIN {X 0,Y 270.743,Z 316.757,A -85,B 0,C 180,E1 -17638.512,E2 -17638.512} C_VEL
LIN {X 0,Y 270.744,Z 316.759,A -85,B 0,C 180,E1 -17641.487,E2 -17641.487} C_VEL
LIN {X 0,Y 270.562,Z 316.772,A -85,B 0,C 180,E1 -17647.463,E2 -17647.463} C_VEL
LIN {X 0,Y 270.4,Z 316.803,A -85,B 0,C 180,E1 -17650.483,E2 -17650.483} C_VEL
LIN {X 0,Y 270.343,Z 316.805,A -85,B 0,C 180,E1 -17655.068,E2 -17655.068} C_VEL
LIN {X 0,Y 270.289,Z 316.806,A -85,B 0,C 180,E1 -17659.757,E2 -17659.757} C_VEL
LIN {X 0,Y 270.248,Z 316.808,A -85,B 0,C 180,E1 -17664.588,E2 -17664.588} C_VEL
LIN {X 0,Y 270.236,Z 316.812,A -85,B 0,C 180,E1 -17667.913,E2 -17667.913} C_VEL
LIN {X 0,Y 270.151,Z 316.827,A -85,B 0,C 180,E1 -17671.353,E2 -17671.353} C_VEL
LIN {X 0,Y 270.189,Z 316.824,A -85,B 0,C 180,E1 -17674.907,E2 -17674.907} C_VEL
LIN {X 0,Y 270.224,Z 316.821,A -85,B 0,C 180,E1 -17678.73,E2 -17678.73} C_VEL
LIN {X 0,Y 270.23,Z 316.83,A -85,B 0,C 180,E1 -17682.547,E2 -17682.547} C_VEL
LIN {X 0,Y 270.208,Z 316.832,A -85,B 0,C 180,E1 -17686.742,E2 -17686.742} C_VEL
LIN {X 0,Y 270.224,Z 316.862,A -85,B 0,C 180,E1 -17690.759,E2 -17690.759} C_VEL
LIN {X 0,Y 272.523,Z 324.848,A -85,B 0,C 180,E1 -17694.087,E2 -17694.087} C_VEL
LIN {X 0,Y 274.841,Z 334.53,A -85,B 0,C 180,E1 -17697.718,E2 -17697.718} C_VEL
LIN {X 0,Y 281.705,Z 349.043,A -85,B 0,C 180,E1 -17699.276,E2 -17699.276} C_VEL
LIN {X 0,Y 284.378,Z 355.71,A -85,B 0,C 180,E1 -17699.88,E2 -17699.88} C_VEL
LIN {X 0,Y 287.738,Z 376.408,A -85,B 0,C 180,E1 -17701.008,E2 -17701.008} C_VEL
LIN {X 0,Y 288.858,Z 386.085,A -85,B 0,C 180,E1 -17701.463,E2 -17701.463} C_VEL
LIN {X 0,Y 286.423,Z 444.91,A -85,B 0,C 180,E1 -17703.06,E2 -17703.06} C_VEL
LIN {X 0,Y 285.169,Z 458.957,A -85,B 0,C 180,E1 -17703.722,E2 -17703.722} C_VEL
LIN {X 0,Y 283.706,Z 470.454,A -85,B 0,C 180,E1 -17704.513,E2 -17704.513} C_VEL
LIN {X 0,Y 281.914,Z 481.508,A -85,B 0,C 180,E1 -17705.522,E2 -17705.522} C_VEL
LIN {X 0,Y 279.812,Z 493.057,A -85,B 0,C 180,E1 -17706.9,E2 -17706.9} C_VEL
LIN {X 0,Y 277.642,Z 503.506,A -85,B 0,C 180,E1 -17708.473,E2 -17708.473} C_VEL
LIN {X 0,Y 275.523,Z 512.961,A -85,B 0,C 180,E1 -17710.253,E2 -17710.253} C_VEL
LIN {X 0,Y 273.443,Z 522.105,A -85,B 0,C 180,E1 -17712.429,E2 -17712.429} C_VEL
LIN {X 0,Y 271.69,Z 529.509,A -85,B 0,C 180,E1 -17714.631,E2 -17714.631} C_VEL
LIN {X 0,Y 270.017,Z 536.338,A -85,B 0,C 180,E1 -17717.224,E2 -17717.224} C_VEL
LIN {X 0,Y 269.141,Z 540.88,A -85,B 0,C 180,E1 -17719.473,E2 -17719.473} C_VEL
LIN {X 0,Y 268.716,Z 543.293,A -85,B 0,C 180,E1 -17720.977,E2 -17720.977} C_VEL
LIN {X 0,Y 268.413,Z 545.277,A -85,B 0,C 180,E1 -17722.483,E2 -17722.483} C_VEL
LIN {X 0,Y 268.174,Z 547.46,A -85,B 0,C 180,E1 -17724.786,E2 -17724.786} C_VEL
LIN {X 0,Y 268.192,Z 548.651,A -85,B 0,C 180,E1 -17727.001,E2 -17727.001} C_VEL
LIN {X 0,Y 268.219,Z 548.973,A -85,B 0,C 180,E1 -17728.504,E2 -17728.504} C_VEL
LIN {X 0,Y 268.252,Z 548.888,A -85,B 0,C 180,E1 -17730.005,E2 -17730.005} C_VEL
LIN {X 0,Y 268.23,Z 548.357,A -85,B 0,C 180,E1 -17731.506,E2 -17731.506} C_VEL
LIN {X 0,Y 268.222,Z 547.425,A -85,B 0,C 180,E1 -17733.009,E2 -17733.009} C_VEL
LIN {X 0,Y 268.196,Z 545.23,A -85,B 0,C 180,E1 -17735.264,E2 -17735.264} C_VEL
LIN {X 0,Y 268.422,Z 542.02,A -85,B 0,C 180,E1 -17737.527,E2 -17737.527} C_VEL
LIN {X 0,Y 268.826,Z 537.712,A -85,B 0,C 180,E1 -17739.788,E2 -17739.788} C_VEL
LIN {X 0,Y 269.677,Z 531.162,A -85,B 0,C 180,E1 -17742.42,E2 -17742.42} C_VEL
LIN {X 0,Y 270.882,Z 523.956,A -85,B 0,C 180,E1 -17744.657,E2 -17744.657} C_VEL
LIN {X 0,Y 272.29,Z 515.491,A -85,B 0,C 180,E1 -17746.759,E2 -17746.759} C_VEL
LIN {X 0,Y 273.756,Z 505.702,A -85,B 0,C 180,E1 -17748.721,E2 -17748.721} C_VEL
LIN {X 0,Y 275.403,Z 495.432,A -85,B 0,C 180,E1 -17750.35,E2 -17750.35} C_VEL
LIN {X 0,Y 277.04,Z 484.045,A -85,B 0,C 180,E1 -17751.781,E2 -17751.781} C_VEL
LIN {X 0,Y 278.525,Z 472.263,A -85,B 0,C 180,E1 -17752.929,E2 -17752.929} C_VEL
LIN {X 0,Y 279.845,Z 459.407,A -85,B 0,C 180,E1 -17753.843,E2 -17753.843} C_VEL
LIN {X 0,Y 280.835,Z 445.886,A -85,B 0,C 180,E1 -17754.49,E2 -17754.49} C_VEL
LIN {X 0,Y 282.758,Z 384.44,A -85,B 0,C 180,E1 -17756.157,E2 -17756.157} C_VEL
LIN {X 0,Y 278.69,Z 354.408,A -85,B 0,C 180,E1 -17757.387,E2 -17757.387} C_VEL
LIN {X 0,Y 276.711,Z 342.909,A -85,B 0,C 180,E1 -17757.911,E2 -17757.911} C_VEL
LIN {X 0,Y 274.528,Z 336.724,A -85,B 0,C 180,E1 -17758.315,E2 -17758.315} C_VEL
LIN {X 0,Y 271.934,Z 324.377,A -85,B 0,C 180,E1 -17762.527,E2 -17762.527} C_VEL
LIN {X 0,Y 270.239,Z 316.823,A -85,B 0,C 180,E1 -17765.244,E2 -17765.244} C_VEL
LIN {X 0,Y 270.205,Z 316.825,A -85,B 0,C 180,E1 -17768.712,E2 -17768.712} C_VEL
LIN {X 0,Y 270.172,Z 316.83,A -85,B 0,C 180,E1 -17773.25,E2 -17773.25} C_VEL
LIN {X 0,Y 270.178,Z 316.83,A -85,B 0,C 180,E1 -17777.443,E2 -17777.443} C_VEL
LIN {X 0,Y 270.214,Z 316.824,A -85,B 0,C 180,E1 -17781.375,E2 -17781.375} C_VEL
LIN {X 0,Y 270.203,Z 316.826,A -85,B 0,C 180,E1 -17785.095,E2 -17785.095} C_VEL
LIN {X 0,Y 270.19,Z 316.827,A -85,B 0,C 180,E1 -17789.137,E2 -17789.137} C_VEL
LIN {X 0,Y 270.268,Z 316.818,A -85,B 0,C 180,E1 -17792.147,E2 -17792.147} C_VEL
LIN {X 0,Y 270.241,Z 316.82,A -85,B 0,C 180,E1 -17795.539,E2 -17795.539} C_VEL
LIN {X 0,Y 270.227,Z 316.819,A -85,B 0,C 180,E1 -17800.239,E2 -17800.239} C_VEL
LIN {X 0,Y 270.37,Z 316.793,A -85,B 0,C 180,E1 -17804.934,E2 -17804.934} C_VEL
LIN {X 0,Y 270.409,Z 316.802,A -85,B 0,C 180,E1 -17809.518,E2 -17809.518} C_VEL
LIN {X 0,Y 270.596,Z 316.774,A -85,B 0,C 180,E1 -17812.538,E2 -17812.538} C_VEL
LIN {X 0,Y 270.785,Z 316.734,A -85,B 0,C 180,E1 -17818.513,E2 -17818.513} C_VEL
LIN {X 0,Y 270.784,Z 316.747,A -85,B 0,C 180,E1 -17821.487,E2 -17821.487} C_VEL
LIN {X 0,Y 270.554,Z 316.784,A -85,B 0,C 180,E1 -17827.463,E2 -17827.463} C_VEL
LIN {X 0,Y 270.389,Z 316.797,A -85,B 0,C 180,E1 -17830.483,E2 -17830.483} C_VEL
LIN {X 0,Y 270.371,Z 316.804,A -85,B 0,C 180,E1 -17835.067,E2 -17835.067} C_VEL
LIN {X 0,Y 270.226,Z 316.819,A -85,B 0,C 180,E1 -17839.761,E2 -17839.761} C_VEL
LIN {X 0,Y 270.187,Z 316.827,A -85,B 0,C 180,E1 -17844.435,E2 -17844.435} C_VEL
LIN {X 0,Y 270.188,Z 316.822,A -85,B 0,C 180,E1 -17847.918,E2 -17847.918} C_VEL
LIN {X 0,Y 270.166,Z 316.808,A -85,B 0,C 180,E1 -17851.351,E2 -17851.351} C_VEL
LIN {X 0,Y 270.199,Z 316.821,A -85,B 0,C 180,E1 -17854.906,E2 -17854.906} C_VEL
LIN {X 0,Y 270.174,Z 316.831,A -85,B 0,C 180,E1 -17858.701,E2 -17858.701} C_VEL
LIN {X 0,Y 270.133,Z 316.831,A -85,B 0,C 180,E1 -17863.239,E2 -17863.239} C_VEL
LIN {X 0,Y 270.135,Z 316.833,A -85,B 0,C 180,E1 -17867.432,E2 -17867.432} C_VEL
LIN {X 0,Y 270.156,Z 316.832,A -85,B 0,C 180,E1 -17871.362,E2 -17871.362} C_VEL
LIN {X 0,Y 270.19,Z 316.827,A -85,B 0,C 180,E1 -17875.09,E2 -17875.09} C_VEL
LIN {X 0,Y 270.176,Z 316.832,A -85,B 0,C 180,E1 -17879.14,E2 -17879.14} C_VEL
LIN {X 0,Y 270.205,Z 316.825,A -85,B 0,C 180,E1 -17882.171,E2 -17882.171} C_VEL
LIN {X 0,Y 270.234,Z 316.822,A -85,B 0,C 180,E1 -17885.54,E2 -17885.54} C_VEL
LIN {X 0,Y 270.231,Z 316.822,A -85,B 0,C 180,E1 -17890.235,E2 -17890.235} C_VEL
LIN {X 0,Y 270.374,Z 316.806,A -85,B 0,C 180,E1 -17894.93,E2 -17894.93} C_VEL
LIN {X 0,Y 270.415,Z 316.802,A -85,B 0,C 180,E1 -17899.514,E2 -17899.514} C_VEL
LIN {X 0,Y 270.566,Z 316.779,A -85,B 0,C 180,E1 -17902.533,E2 -17902.533} C_VEL
LIN {X 0,Y 270.777,Z 316.753,A -85,B 0,C 180,E1 -17908.508,E2 -17908.508} C_VEL
LIN {X 0,Y 270.674,Z 316.768,A -85,B 0,C 180,E1 -17912.227,E2 -17912.227} C_VEL
LIN {X 0,Y 270.618,Z 316.94,A -85,B 0,C 180,E1 -17912.972,E2 -17912.972} C_VEL
LIN {X 0,Y 270.876,Z 318.386,A -85,B 0,C 180,E1 -17913.434,E2 -17913.434} C_VEL
LIN {X 0,Y 279.6,Z 340.537,A -85,B 0,C 180,E1 -17914.918,E2 -17914.918} C_VEL
LIN {X 0,Y 283.487,Z 351.733,A -85,B 0,C 180,E1 -17915.588,E2 -17915.588} C_VEL
LIN {X 0,Y 281.138,Z 425.736,A -85,B 0,C 180,E1 -17917.581,E2 -17917.581} C_VEL
LIN {X 0,Y 280.334,Z 439.251,A -85,B 0,C 180,E1 -17918.238,E2 -17918.238} C_VEL
LIN {X 0,Y 279.34,Z 451.65,A -85,B 0,C 180,E1 -17919.126,E2 -17919.126} C_VEL
LIN {X 0,Y 278.076,Z 462.74,A -85,B 0,C 180,E1 -17920.185,E2 -17920.185} C_VEL
LIN {X 0,Y 276.562,Z 473.812,A -85,B 0,C 180,E1 -17921.538,E2 -17921.538} C_VEL
LIN {X 0,Y 275.009,Z 484.021,A -85,B 0,C 180,E1 -17923.103,E2 -17923.103} C_VEL
LIN {X 0,Y 273.578,Z 493.359,A -85,B 0,C 180,E1 -17924.88,E2 -17924.88} C_VEL
LIN {X 0,Y 272.013,Z 502.531,A -85,B 0,C 180,E1 -17927.065,E2 -17927.065} C_VEL
LIN {X 0,Y 270.773,Z 510.067,A -85,B 0,C 180,E1 -17929.319,E2 -17929.319} C_VEL
LIN {X 0,Y 269.911,Z 515.562,A -85,B 0,C 180,E1 -17931.372,E2 -17931.372} C_VEL
LIN {X 0,Y 269.121,Z 520.938,A -85,B 0,C 180,E1 -17933.934,E2 -17933.934} C_VEL
LIN {X 0,Y 268.499,Z 524.733,A -85,B 0,C 180,E1 -17936.414,E2 -17936.414} C_VEL
LIN {X 0,Y 268.159,Z 526.653,A -85,B 0,C 180,E1 -17938.14,E2 -17938.14} C_VEL
LIN {X 0,Y 267.984,Z 528.137,A -85,B 0,C 180,E1 -17940.067,E2 -17940.067} C_VEL
LIN {X 0,Y 267.963,Z 529.116,A -85,B 0,C 180,E1 -17942.936,E2 -17942.936} C_VEL
LIN {X 0,Y 268.223,Z 528.706,A -85,B 0,C 180,E1 -17945.682,E2 -17945.682} C_VEL
LIN {X 0,Y 268.731,Z 527.017,A -85,B 0,C 180,E1 -17948.318,E2 -17948.318} C_VEL
LIN {X 0,Y 269.514,Z 524.16,A -85,B 0,C 180,E1 -17950.867,E2 -17950.867} C_VEL
LIN {X 0,Y 270.566,Z 520.154,A -85,B 0,C 180,E1 -17953.339,E2 -17953.339} C_VEL
LIN {X 0,Y 271.93,Z 514.918,A -85,B 0,C 180,E1 -17955.748,E2 -17955.748} C_VEL
LIN {X 0,Y 273.664,Z 508.215,A -85,B 0,C 180,E1 -17958.126,E2 -17958.126} C_VEL
LIN {X 0,Y 275.781,Z 499.864,A -85,B 0,C 180,E1 -17960.424,E2 -17960.424} C_VEL
LIN {X 0,Y 277.99,Z 490.418,A -85,B 0,C 180,E1 -17962.486,E2 -17962.486} C_VEL
LIN {X 0,Y 279.804,Z 481.462,A -85,B 0,C 180,E1 -17964.06,E2 -17964.06} C_VEL
LIN {X 0,Y 282.024,Z 470.169,A -85,B 0,C 180,E1 -17965.622,E2 -17965.622} C_VEL
LIN {X 0,Y 283.827,Z 458.775,A -85,B 0,C 180,E1 -17966.868,E2 -17966.868} C_VEL
LIN {X 0,Y 285.325,Z 447.114,A -85,B 0,C 180,E1 -17967.841,E2 -17967.841} C_VEL
LIN {X 0,Y 286.423,Z 434.443,A -85,B 0,C 180,E1 -17968.614,E2 -17968.614} C_VEL
LIN {X 0,Y 287.335,Z 421.393,A -85,B 0,C 180,E1 -17969.105,E2 -17969.105} C_VEL
LIN {X 0,Y 289.828,Z 357.043,A -85,B 0,C 180,E1 -17970.83,E2 -17970.83} C_VEL
LIN {X 0,Y 283.732,Z 343.042,A -85,B 0,C 180,E1 -17972.126,E2 -17972.126} C_VEL
LIN {X 0,Y 277.344,Z 330.405,A -85,B 0,C 180,E1 -17973.523,E2 -17973.523} C_VEL
LIN {X 0,Y 272.229,Z 321.701,A -85,B 0,C 180,E1 -17974.663,E2 -17974.663} C_VEL
LIN {X 0,Y 270.892,Z 319.092,A -85,B 0,C 180,E1 -17974.993,E2 -17974.993} C_VEL
LIN {X 0,Y 270.222,Z 316.834,A -85,B 0,C 180,E1 -17976.027,E2 -17976.027} C_VEL
LIN {X 0,Y 270.226,Z 316.833,A -85,B 0,C 180,E1 -17976.099,E2 -17976.099} C_VEL
LIN {X 0,Y 269.532,Z 316.919,A -85,B 0,C 180,E1 -17977.343,E2 -17977.343} C_VEL
LIN {X 0,Y 266.653,Z 317.274,A -85,B 0,C 180,E1 -17979.37,E2 -17979.37} C_VEL
LIN {X 0,Y 264.251,Z 317.569,A -85,B 0,C 180,E1 -17981.018,E2 -17981.018} C_VEL
LIN {X 0,Y 263.26,Z 317.696,A -85,B 0,C 180,E1 -17982.295,E2 -17982.295} C_VEL
LIN {X 0,Y 263.199,Z 317.7,A -85,B 0,C 180,E1 -17982.728,E2 -17982.728} C_VEL
LIN {X 0,Y 263.253,Z 317.69,A -85,B 0,C 180,E1 -17986.097,E2 -17986.097} C_VEL
LIN {X 0,Y 263.432,Z 317.671,A -85,B 0,C 180,E1 -17990.789,E2 -17990.789} C_VEL
LIN {X 0,Y 263.464,Z 317.665,A -85,B 0,C 180,E1 -17993.875,E2 -17993.875} C_VEL
LIN {X 0,Y 263.708,Z 317.634,A -85,B 0,C 180,E1 -17998.473,E2 -17998.473} C_VEL
LIN {X 0,Y 263.708,Z 317.636,A -85,B 0,C 180,E1 -18001.527,E2 -18001.527} C_VEL
LIN {X 0,Y 263.524,Z 317.648,A -85,B 0,C 180,E1 -18007.663,E2 -18007.663} C_VEL
LIN {X 0,Y 263.333,Z 317.68,A -85,B 0,C 180,E1 -18010.767,E2 -18010.767} C_VEL
LIN {X 0,Y 263.29,Z 317.679,A -85,B 0,C 180,E1 -18015.482,E2 -18015.482} C_VEL
LIN {X 0,Y 263.252,Z 317.679,A -85,B 0,C 180,E1 -18020.308,E2 -18020.308} C_VEL
LIN {X 0,Y 263.178,Z 317.692,A -85,B 0,C 180,E1 -18025.294,E2 -18025.294} C_VEL
LIN {X 0,Y 263.142,Z 317.696,A -85,B 0,C 180,E1 -18028.734,E2 -18028.734} C_VEL
LIN {X 0,Y 263.101,Z 317.705,A -85,B 0,C 180,E1 -18032.293,E2 -18032.293} C_VEL
LIN {X 0,Y 263.166,Z 317.7,A -85,B 0,C 180,E1 -18035.982,E2 -18035.982} C_VEL
LIN {X 0,Y 263.174,Z 317.707,A -85,B 0,C 180,E1 -18039.86,E2 -18039.86} C_VEL
LIN {X 0,Y 263.165,Z 317.706,A -85,B 0,C 180,E1 -18043.975,E2 -18043.975} C_VEL
LIN {X 0,Y 263.189,Z 317.704,A -85,B 0,C 180,E1 -18048.391,E2 -18048.391} C_VEL
LIN {X 0,Y 263.193,Z 317.707,A -85,B 0,C 180,E1 -18049.653,E2 -18049.653} C_VEL
LIN {X 0,Y 265.714,Z 326.598,A -85,B 0,C 180,E1 -18053.53,E2 -18053.53} C_VEL
LIN {X 0,Y 267.547,Z 334.009,A -85,B 0,C 180,E1 -18056.477,E2 -18056.477} C_VEL
LIN {X 0,Y 274.858,Z 348.982,A -85,B 0,C 180,E1 -18058.233,E2 -18058.233} C_VEL
LIN {X 0,Y 278.661,Z 357.747,A -85,B 0,C 180,E1 -18059.123,E2 -18059.123} C_VEL
LIN {X 0,Y 281.913,Z 378.126,A -85,B 0,C 180,E1 -18060.275,E2 -18060.275} C_VEL
LIN {X 0,Y 282.895,Z 387.032,A -85,B 0,C 180,E1 -18060.702,E2 -18060.702} C_VEL
LIN {X 0,Y 280.442,Z 444.265,A -85,B 0,C 180,E1 -18062.285,E2 -18062.285} C_VEL
LIN {X 0,Y 279.131,Z 458.381,A -85,B 0,C 180,E1 -18062.956,E2 -18062.956} C_VEL
LIN {X 0,Y 277.517,Z 470.457,A -85,B 0,C 180,E1 -18063.801,E2 -18063.801} C_VEL
LIN {X 0,Y 275.522,Z 482.194,A -85,B 0,C 180,E1 -18064.915,E2 -18064.915} C_VEL
LIN {X 0,Y 273.335,Z 493.541,A -85,B 0,C 180,E1 -18066.319,E2 -18066.319} C_VEL
LIN {X 0,Y 271.072,Z 503.847,A -85,B 0,C 180,E1 -18067.925,E2 -18067.925} C_VEL
LIN {X 0,Y 268.864,Z 513.162,A -85,B 0,C 180,E1 -18069.742,E2 -18069.742} C_VEL
LIN {X 0,Y 266.688,Z 522.228,A -85,B 0,C 180,E1 -18071.969,E2 -18071.969} C_VEL
LIN {X 0,Y 264.848,Z 529.566,A -85,B 0,C 180,E1 -18074.223,E2 -18074.223} C_VEL
LIN {X 0,Y 263.5,Z 534.549,A -85,B 0,C 180,E1 -18076.117,E2 -18076.117} C_VEL
LIN {X 0,Y 262.404,Z 539.415,A -85,B 0,C 180,E1 -18078.418,E2 -18078.418} C_VEL
LIN {X 0,Y 261.69,Z 543.172,A -85,B 0,C 180,E1 -18080.733,E2 -18080.733} C_VEL
LIN {X 0,Y 261.347,Z 545.129,A -85,B 0,C 180,E1 -18082.278,E2 -18082.278} C_VEL
LIN {X 0,Y 261.083,Z 547.432,A -85,B 0,C 180,E1 -18084.868,E2 -18084.868} C_VEL
LIN {X 0,Y 261.104,Z 548.416,A -85,B 0,C 180,E1 -18086.919,E2 -18086.919} C_VEL
LIN {X 0,Y 261.144,Z 548.718,A -85,B 0,C 180,E1 -18088.463,E2 -18088.463} C_VEL
LIN {X 0,Y 261.176,Z 548.592,A -85,B 0,C 180,E1 -18090.005,E2 -18090.005} C_VEL
LIN {X 0,Y 261.156,Z 548.039,A -85,B 0,C 180,E1 -18091.547,E2 -18091.547} C_VEL
LIN {X 0,Y 261.132,Z 547.084,A -85,B 0,C 180,E1 -18093.09,E2 -18093.09} C_VEL
LIN {X 0,Y 261.126,Z 545.045,A -85,B 0,C 180,E1 -18095.235,E2 -18095.235} C_VEL
LIN {X 0,Y 261.352,Z 541.584,A -85,B 0,C 180,E1 -18097.732,E2 -18097.732} C_VEL
LIN {X 0,Y 261.781,Z 537.223,A -85,B 0,C 180,E1 -18100.054,E2 -18100.054} C_VEL
LIN {X 0,Y 262.514,Z 531.639,A -85,B 0,C 180,E1 -18102.371,E2 -18102.371} C_VEL
LIN {X 0,Y 263.748,Z 524.661,A -85,B 0,C 180,E1 -18104.668,E2 -18104.668} C_VEL
LIN {X 0,Y 265.001,Z 517.514,A -85,B 0,C 180,E1 -18106.569,E2 -18106.569} C_VEL
LIN {X 0,Y 266.38,Z 508.844,A -85,B 0,C 180,E1 -18108.461,E2 -18108.461} C_VEL
LIN {X 0,Y 268.035,Z 498.141,A -85,B 0,C 180,E1 -18110.333,E2 -18110.333} C_VEL
LIN {X 0,Y 269.764,Z 487.566,A -85,B 0,C 180,E1 -18111.796,E2 -18111.796} C_VEL
LIN {X 0,Y 271.357,Z 475.849,A -85,B 0,C 180,E1 -18113.066,E2 -18113.066} C_VEL
LIN {X 0,Y 272.864,Z 462.452,A -85,B 0,C 180,E1 -18114.138,E2 -18114.138} C_VEL
LIN {X 0,Y 273.944,Z 449.751,A -85,B 0,C 180,E1 -18114.844,E2 -18114.844} C_VEL
LIN {X 0,Y 274.601,Z 434.998,A -85,B 0,C 180,E1 -18115.337,E2 -18115.337} C_VEL
LIN {X 0,Y 276.134,Z 384.453,A -85,B 0,C 180,E1 -18116.714,E2 -18116.714} C_VEL
LIN {X 0,Y 271.925,Z 353.942,A -85,B 0,C 180,E1 -18118.015,E2 -18118.015} C_VEL
LIN {X 0,Y 270.411,Z 345.281,A -85,B 0,C 180,E1 -18118.423,E2 -18118.423} C_VEL
LIN {X 0,Y 267.238,Z 336.347,A -85,B 0,C 180,E1 -18119.049,E2 -18119.049} C_VEL
LIN {X 0,Y 264.879,Z 325.265,A -85,B 0,C 180,E1 -18122.953,E2 -18122.953} C_VEL
LIN {X 0,Y 263.201,Z 317.702,A -85,B 0,C 180,E1 -18125.762,E2 -18125.762} C_VEL
LIN {X 0,Y 263.113,Z 317.709,A -85,B 0,C 180,E1 -18129.874,E2 -18129.874} C_VEL
LIN {X 0,Y 263.111,Z 317.711,A -85,B 0,C 180,E1 -18133.99,E2 -18133.99} C_VEL
LIN {X 0,Y 263.131,Z 317.71,A -85,B 0,C 180,E1 -18138.408,E2 -18138.408} C_VEL
LIN {X 0,Y 263.164,Z 317.704,A -85,B 0,C 180,E1 -18142.104,E2 -18142.104} C_VEL
LIN {X 0,Y 263.158,Z 317.703,A -85,B 0,C 180,E1 -18145.886,E2 -18145.886} C_VEL
LIN {X 0,Y 263.135,Z 317.704,A -85,B 0,C 180,E1 -18149.505,E2 -18149.505} C_VEL
LIN {X 0,Y 263.195,Z 317.701,A -85,B 0,C 180,E1 -18153.003,E2 -18153.003} C_VEL
LIN {X 0,Y 263.156,Z 317.702,A -85,B 0,C 180,E1 -18156.384,E2 -18156.384} C_VEL
LIN {X 0,Y 263.213,Z 317.693,A -85,B 0,C 180,E1 -18159.689,E2 -18159.689} C_VEL
LIN {X 0,Y 263.313,Z 317.669,A -85,B 0,C 180,E1 -18164.52,E2 -18164.52} C_VEL
LIN {X 0,Y 263.349,Z 317.682,A -85,B 0,C 180,E1 -18169.233,E2 -18169.233} C_VEL
LIN {X 0,Y 263.557,Z 317.651,A -85,B 0,C 180,E1 -18172.338,E2 -18172.338} C_VEL
LIN {X 0,Y 263.75,Z 317.608,A -85,B 0,C 180,E1 -18178.473,E2 -18178.473} C_VEL
LIN {X 0,Y 263.749,Z 317.623,A -85,B 0,C 180,E1 -18181.527,E2 -18181.527} C_VEL
LIN {X 0,Y 263.516,Z 317.66,A -85,B 0,C 180,E1 -18187.663,E2 -18187.663} C_VEL
LIN {X 0,Y 263.336,Z 317.675,A -85,B 0,C 180,E1 -18190.767,E2 -18190.767} C_VEL
LIN {X 0,Y 263.314,Z 317.685,A -85,B 0,C 180,E1 -18195.48,E2 -18195.48} C_VEL
LIN {X 0,Y 263.212,Z 317.695,A -85,B 0,C 180,E1 -18200.311,E2 -18200.311} C_VEL
LIN {X 0,Y 263.108,Z 317.707,A -85,B 0,C 180,E1 -18205.302,E2 -18205.302} C_VEL
LIN {X 0,Y 263.122,Z 317.694,A -85,B 0,C 180,E1 -18208.737,E2 -18208.737} C_VEL
LIN {X 0,Y 263.121,Z 317.688,A -85,B 0,C 180,E1 -18212.29,E2 -18212.29} C_VEL
LIN {X 0,Y 263.157,Z 317.699,A -85,B 0,C 180,E1 -18215.983,E2 -18215.983} C_VEL
LIN {X 0,Y 263.076,Z 317.713,A -85,B 0,C 180,E1 -18219.878,E2 -18219.878} C_VEL
LIN {X 0,Y 263.077,Z 317.71,A -85,B 0,C 180,E1 -18223.994,E2 -18223.994} C_VEL
LIN {X 0,Y 263.07,Z 317.714,A -85,B 0,C 180,E1 -18228.093,E2 -18228.093} C_VEL
LIN {X 0,Y 263.106,Z 317.71,A -85,B 0,C 180,E1 -18232.091,E2 -18232.091} C_VEL
LIN {X 0,Y 263.159,Z 317.7,A -85,B 0,C 180,E1 -18235.883,E2 -18235.883} C_VEL
LIN {X 0,Y 263.115,Z 317.71,A -85,B 0,C 180,E1 -18239.499,E2 -18239.499} C_VEL
LIN {X 0,Y 263.137,Z 317.711,A -85,B 0,C 180,E1 -18242.993,E2 -18242.993} C_VEL
LIN {X 0,Y 263.151,Z 317.704,A -85,B 0,C 180,E1 -18246.38,E2 -18246.38} C_VEL
LIN {X 0,Y 263.216,Z 317.697,A -85,B 0,C 180,E1 -18249.686,E2 -18249.686} C_VEL
LIN {X 0,Y 263.317,Z 317.683,A -85,B 0,C 180,E1 -18254.516,E2 -18254.516} C_VEL
LIN {X 0,Y 263.355,Z 317.681,A -85,B 0,C 180,E1 -18259.229,E2 -18259.229} C_VEL
LIN {X 0,Y 263.53,Z 317.656,A -85,B 0,C 180,E1 -18262.333,E2 -18262.333} C_VEL
LIN {X 0,Y 263.74,Z 317.63,A -85,B 0,C 180,E1 -18268.468,E2 -18268.468} C_VEL
LIN {X 0,Y 263.639,Z 317.643,A -85,B 0,C 180,E1 -18272.382,E2 -18272.382} C_VEL
LIN {X 0,Y 263.725,Z 318.385,A -85,B 0,C 180,E1 -18272.716,E2 -18272.716} C_VEL
LIN {X 0,Y 273.433,Z 343.169,A -85,B 0,C 180,E1 -18274.436,E2 -18274.436} C_VEL
LIN {X 0,Y 276.888,Z 353.157,A -85,B 0,C 180,E1 -18275.05,E2 -18275.05} C_VEL
LIN {X 0,Y 274.542,Z 425.531,A -85,B 0,C 180,E1 -18277.044,E2 -18277.044} C_VEL
LIN {X 0,Y 273.722,Z 438.883,A -85,B 0,C 180,E1 -18277.695,E2 -18277.695} C_VEL
LIN {X 0,Y 272.663,Z 451.558,A -85,B 0,C 180,E1 -18278.611,E2 -18278.611} C_VEL
LIN {X 0,Y 271.288,Z 463.429,A -85,B 0,C 180,E1 -18279.774,E2 -18279.774} C_VEL
LIN {X 0,Y 269.636,Z 475.179,A -85,B 0,C 180,E1 -18281.267,E2 -18281.267} C_VEL
LIN {X 0,Y 268.038,Z 485.21,A -85,B 0,C 180,E1 -18282.872,E2 -18282.872} C_VEL
LIN {X 0,Y 266.405,Z 495.253,A -85,B 0,C 180,E1 -18284.899,E2 -18284.899} C_VEL
LIN {X 0,Y 264.824,Z 504.268,A -85,B 0,C 180,E1 -18287.179,E2 -18287.179} C_VEL
LIN {X 0,Y 263.624,Z 511.414,A -85,B 0,C 180,E1 -18289.459,E2 -18289.459} C_VEL
LIN {X 0,Y 262.571,Z 517.641,A -85,B 0,C 180,E1 -18292,E2 -18292} C_VEL
LIN {X 0,Y 261.971,Z 521.828,A -85,B 0,C 180,E1 -18294.198,E2 -18294.198} C_VEL
LIN {X 0,Y 261.419,Z 524.952,A -85,B 0,C 180,E1 -18296.325,E2 -18296.325} C_VEL
LIN {X 0,Y 260.955,Z 527.641,A -85,B 0,C 180,E1 -18298.99,E2 -18298.99} C_VEL
LIN {X 0,Y 260.837,Z 528.77,A -85,B 0,C 180,E1 -18300.785,E2 -18300.785} C_VEL
LIN {X 0,Y 260.893,Z 529.423,A -85,B 0,C 180,E1 -18303.375,E2 -18303.375} C_VEL
LIN {X 0,Y 261.205,Z 528.79,A -85,B 0,C 180,E1 -18306.285,E2 -18306.285} C_VEL
LIN {X 0,Y 261.769,Z 527.045,A -85,B 0,C 180,E1 -18308.868,E2 -18308.868} C_VEL
LIN {X 0,Y 262.871,Z 523.459,A -85,B 0,C 180,E1 -18311.933,E2 -18311.933} C_VEL
LIN {X 0,Y 264.235,Z 518.329,A -85,B 0,C 180,E1 -18314.826,E2 -18314.826} C_VEL
LIN {X 0,Y 265.639,Z 513.209,A -85,B 0,C 180,E1 -18317.007,E2 -18317.007} C_VEL
LIN {X 0,Y 267.773,Z 505.557,A -85,B 0,C 180,E1 -18319.552,E2 -18319.552} C_VEL
LIN {X 0,Y 269.889,Z 497.434,A -85,B 0,C 180,E1 -18321.658,E2 -18321.658} C_VEL
LIN {X 0,Y 272.029,Z 488.425,A -85,B 0,C 180,E1 -18323.543,E2 -18323.543} C_VEL
LIN {X 0,Y 274.267,Z 477.956,A -85,B 0,C 180,E1 -18325.302,E2 -18325.302} C_VEL
LIN {X 0,Y 276.43,Z 466.628,A -85,B 0,C 180,E1 -18326.78,E2 -18326.78} C_VEL
LIN {X 0,Y 278.247,Z 454.955,A -85,B 0,C 180,E1 -18327.966,E2 -18327.966} C_VEL
LIN {X 0,Y 279.639,Z 443.408,A -85,B 0,C 180,E1 -18328.858,E2 -18328.858} C_VEL
LIN {X 0,Y 280.745,Z 430.79,A -85,B 0,C 180,E1 -18329.544,E2 -18329.544} C_VEL
LIN {X 0,Y 281.676,Z 413.363,A -85,B 0,C 180,E1 -18330.093,E2 -18330.093} C_VEL
LIN {X 0,Y 283.884,Z 359.015,A -85,B 0,C 180,E1 -18331.575,E2 -18331.575} C_VEL
LIN {X 0,Y 277.22,Z 343.848,A -85,B 0,C 180,E1 -18333.072,E2 -18333.072} C_VEL
LIN {X 0,Y 270.566,Z 331.206,A -85,B 0,C 180,E1 -18334.596,E2 -18334.596} C_VEL
LIN {X 0,Y 265.666,Z 323.064,A -85,B 0,C 180,E1 -18335.766,E2 -18335.766} C_VEL
LIN {X 0,Y 263.601,Z 319.35,A -85,B 0,C 180,E1 -18336.34,E2 -18336.34} C_VEL
LIN {X 0,Y 263.135,Z 317.714,A -85,B 0,C 180,E1 -18337.111,E2 -18337.111} C_VEL
LIN {X 0,Y 263.224,Z 317.702,A -85,B 0,C 180,E1 -18339.69,E2 -18339.69} C_VEL
LIN {X 0,Y 263.199,Z 317.7,A -85,B 0,C 180,E1 -18342.728,E2 -18342.728} C_VEL
LIN {X 0,Y 262.581,Z 317.783,A -85,B 0,C 180,E1 -18344.006,E2 -18344.006} C_VEL
LIN {X 0,Y 259.741,Z 318.135,A -85,B 0,C 180,E1 -18346.088,E2 -18346.088} C_VEL
LIN {X 0,Y 257.327,Z 318.432,A -85,B 0,C 180,E1 -18347.783,E2 -18347.783} C_VEL
LIN {X 0,Y 256.328,Z 318.55,A -85,B 0,C 180,E1 -18349.097,E2 -18349.097} C_VEL
LIN {X 0,Y 256.269,Z 318.556,A -85,B 0,C 180,E1 -18349.542,E2 -18349.542} C_VEL
LIN {X 0,Y 256.471,Z 318.532,A -85,B 0,C 180,E1 -18352.125,E2 -18352.125} C_VEL
LIN {X 0,Y 256.454,Z 318.533,A -85,B 0,C 180,E1 -18356.858,E2 -18356.858} C_VEL
LIN {X 0,Y 256.714,Z 318.496,A -85,B 0,C 180,E1 -18360,E2 -18360} C_VEL
LIN {X 0,Y 256.456,Z 318.53,A -85,B 0,C 180,E1 -18363.142,E2 -18363.142} C_VEL
LIN {X 0,Y 256.488,Z 318.524,A -85,B 0,C 180,E1 -18367.875,E2 -18367.875} C_VEL
LIN {X 0,Y 256.269,Z 318.556,A -85,B 0,C 180,E1 -18371.068,E2 -18371.068} C_VEL
LIN {X 0,Y 256.226,Z 318.556,A -85,B 0,C 180,E1 -18375.92,E2 -18375.92} C_VEL
LIN {X 0,Y 256.201,Z 318.558,A -85,B 0,C 180,E1 -18380.892,E2 -18380.892} C_VEL
LIN {X 0,Y 256.159,Z 318.565,A -85,B 0,C 180,E1 -18385.144,E2 -18385.144} C_VEL
LIN {X 0,Y 256.078,Z 318.583,A -85,B 0,C 180,E1 -18389.604,E2 -18389.604} C_VEL
LIN {X 0,Y 256.054,Z 318.589,A -85,B 0,C 180,E1 -18393.295,E2 -18393.295} C_VEL
LIN {X 0,Y 256.126,Z 318.581,A -85,B 0,C 180,E1 -18397.288,E2 -18397.288} C_VEL
LIN {X 0,Y 256.137,Z 318.578,A -85,B 0,C 180,E1 -18401.188,E2 -18401.188} C_VEL
LIN {X 0,Y 256.092,Z 318.59,A -85,B 0,C 180,E1 -18405.523,E2 -18405.523} C_VEL
LIN {X 0,Y 256.184,Z 318.695,A -85,B 0,C 180,E1 -18408.5,E2 -18408.5} C_VEL
LIN {X 0,Y 259.004,Z 328.388,A -85,B 0,C 180,E1 -18412.953,E2 -18412.953} C_VEL
LIN {X 0,Y 260.361,Z 333.872,A -85,B 0,C 180,E1 -18415.159,E2 -18415.159} C_VEL
LIN {X 0,Y 266.122,Z 345.163,A -85,B 0,C 180,E1 -18416.647,E2 -18416.647} C_VEL
LIN {X 0,Y 271.674,Z 357.002,A -85,B 0,C 180,E1 -18418.011,E2 -18418.011} C_VEL
LIN {X 0,Y 273.337,Z 361.217,A -85,B 0,C 180,E1 -18418.426,E2 -18418.426} C_VEL
LIN {X 0,Y 276.349,Z 381.583,A -85,B 0,C 180,E1 -18419.598,E2 -18419.598} C_VEL
LIN {X 0,Y 276.967,Z 388.278,A -85,B 0,C 180,E1 -18419.917,E2 -18419.917} C_VEL
LIN {X 0,Y 274.424,Z 444.721,A -85,B 0,C 180,E1 -18421.519,E2 -18421.519} C_VEL
LIN {X 0,Y 273.055,Z 458.597,A -85,B 0,C 180,E1 -18422.2,E2 -18422.2} C_VEL
LIN {X 0,Y 271.376,Z 470.517,A -85,B 0,C 180,E1 -18423.058,E2 -18423.058} C_VEL
LIN {X 0,Y 269.143,Z 482.961,A -85,B 0,C 180,E1 -18424.278,E2 -18424.278} C_VEL
LIN {X 0,Y 266.89,Z 494.122,A -85,B 0,C 180,E1 -18425.711,E2 -18425.711} C_VEL
LIN {X 0,Y 264.528,Z 504.245,A -85,B 0,C 180,E1 -18427.349,E2 -18427.349} C_VEL
LIN {X 0,Y 262.211,Z 513.404,A -85,B 0,C 180,E1 -18429.205,E2 -18429.205} C_VEL
LIN {X 0,Y 259.951,Z 522.363,A -85,B 0,C 180,E1 -18431.484,E2 -18431.484} C_VEL
LIN {X 0,Y 258.022,Z 529.62,A -85,B 0,C 180,E1 -18433.795,E2 -18433.795} C_VEL
LIN {X 0,Y 256.151,Z 536.274,A -85,B 0,C 180,E1 -18436.52,E2 -18436.52} C_VEL
LIN {X 0,Y 255.112,Z 540.702,A -85,B 0,C 180,E1 -18438.887,E2 -18438.887} C_VEL
LIN {X 0,Y 254.643,Z 543.061,A -85,B 0,C 180,E1 -18440.474,E2 -18440.474} C_VEL
LIN {X 0,Y 254.304,Z 544.99,A -85,B 0,C 180,E1 -18442.063,E2 -18442.063} C_VEL
LIN {X 0,Y 253.972,Z 547.513,A -85,B 0,C 180,E1 -18445.244,E2 -18445.244} C_VEL
LIN {X 0,Y 253.999,Z 548.183,A -85,B 0,C 180,E1 -18446.833,E2 -18446.833} C_VEL
LIN {X 0,Y 254.071,Z 548.46,A -85,B 0,C 180,E1 -18448.42,E2 -18448.42} C_VEL
LIN {X 0,Y 254.101,Z 548.292,A -85,B 0,C 180,E1 -18450.005,E2 -18450.005} C_VEL
LIN {X 0,Y 254.083,Z 547.717,A -85,B 0,C 180,E1 -18451.59,E2 -18451.59} C_VEL
LIN {X 0,Y 254.045,Z 546.739,A -85,B 0,C 180,E1 -18453.177,E2 -18453.177} C_VEL
LIN {X 0,Y 254.024,Z 544.946,A -85,B 0,C 180,E1 -18455.123,E2 -18455.123} C_VEL
LIN {X 0,Y 254.308,Z 541.145,A -85,B 0,C 180,E1 -18457.947,E2 -18457.947} C_VEL
LIN {X 0,Y 254.754,Z 536.729,A -85,B 0,C 180,E1 -18460.335,E2 -18460.335} C_VEL
LIN {X 0,Y 255.543,Z 531.085,A -85,B 0,C 180,E1 -18462.714,E2 -18462.714} C_VEL
LIN {X 0,Y 256.842,Z 524.027,A -85,B 0,C 180,E1 -18465.071,E2 -18465.071} C_VEL
LIN {X 0,Y 258.413,Z 515.146,A -85,B 0,C 180,E1 -18467.411,E2 -18467.411} C_VEL
LIN {X 0,Y 260.042,Z 505.028,A -85,B 0,C 180,E1 -18469.543,E2 -18469.543} C_VEL
LIN {X 0,Y 261.805,Z 494.708,A -85,B 0,C 180,E1 -18471.251,E2 -18471.251} C_VEL
LIN {X 0,Y 263.583,Z 483.279,A -85,B 0,C 180,E1 -18472.748,E2 -18472.748} C_VEL
LIN {X 0,Y 265.178,Z 471.431,A -85,B 0,C 180,E1 -18473.947,E2 -18473.947} C_VEL
LIN {X 0,Y 266.544,Z 458.419,A -85,B 0,C 180,E1 -18474.904,E2 -18474.904} C_VEL
LIN {X 0,Y 267.626,Z 444.72,A -85,B 0,C 180,E1 -18475.576,E2 -18475.576} C_VEL
LIN {X 0,Y 269.586,Z 385.179,A -85,B 0,C 180,E1 -18477.266,E2 -18477.266} C_VEL
LIN {X 0,Y 265.405,Z 354.849,A -85,B 0,C 180,E1 -18478.596,E2 -18478.596} C_VEL
LIN {X 0,Y 264.177,Z 347.668,A -85,B 0,C 180,E1 -18478.944,E2 -18478.944} C_VEL
LIN {X 0,Y 259.929,Z 336.155,A -85,B 0,C 180,E1 -18479.764,E2 -18479.764} C_VEL
LIN {X 0,Y 257.762,Z 325.84,A -85,B 0,C 180,E1 -18483.516,E2 -18483.516} C_VEL
LIN {X 0,Y 256.157,Z 318.575,A -85,B 0,C 180,E1 -18486.335,E2 -18486.335} C_VEL
LIN {X 0,Y 256.068,Z 318.586,A -85,B 0,C 180,E1 -18489.782,E2 -18489.782} C_VEL
LIN {X 0,Y 256.056,Z 318.589,A -85,B 0,C 180,E1 -18493.332,E2 -18493.332} C_VEL
LIN {X 0,Y 256.076,Z 318.587,A -85,B 0,C 180,E1 -18497.821,E2 -18497.821} C_VEL
LIN {X 0,Y 256.078,Z 318.588,A -85,B 0,C 180,E1 -18500.859,E2 -18500.859} C_VEL
LIN {X 0,Y 256.133,Z 318.582,A -85,B 0,C 180,E1 -18502.868,E2 -18502.868} C_VEL
LIN {X 0,Y 256.072,Z 318.59,A -85,B 0,C 180,E1 -18506.708,E2 -18506.708} C_VEL
LIN {X 0,Y 256.132,Z 318.58,A -85,B 0,C 180,E1 -18511.411,E2 -18511.411} C_VEL
LIN {X 0,Y 256.146,Z 318.575,A -85,B 0,C 180,E1 -18515.697,E2 -18515.697} C_VEL
LIN {X 0,Y 256.129,Z 318.579,A -85,B 0,C 180,E1 -18519.102,E2 -18519.102} C_VEL
LIN {X 0,Y 256.233,Z 318.548,A -85,B 0,C 180,E1 -18524.081,E2 -18524.081} C_VEL
LIN {X 0,Y 256.29,Z 318.559,A -85,B 0,C 180,E1 -18528.933,E2 -18528.933} C_VEL
LIN {X 0,Y 256.516,Z 318.528,A -85,B 0,C 180,E1 -18532.126,E2 -18532.126} C_VEL
LIN {X 0,Y 256.492,Z 318.516,A -85,B 0,C 180,E1 -18536.859,E2 -18536.859} C_VEL
LIN {X 0,Y 256.745,Z 318.491,A -85,B 0,C 180,E1 -18540,E2 -18540} C_VEL
LIN {X 0,Y 256.489,Z 318.53,A -85,B 0,C 180,E1 -18543.142,E2 -18543.142} C_VEL
LIN {X 0,Y 256.458,Z 318.537,A -85,B 0,C 180,E1 -18547.876,E2 -18547.876} C_VEL
LIN {X 0,Y 256.282,Z 318.553,A -85,B 0,C 180,E1 -18551.067,E2 -18551.067} C_VEL
LIN {X 0,Y 256.235,Z 318.567,A -85,B 0,C 180,E1 -18555.919,E2 -18555.919} C_VEL
LIN {X 0,Y 256.124,Z 318.576,A -85,B 0,C 180,E1 -18561.096,E2 -18561.096} C_VEL
LIN {X 0,Y 256.082,Z 318.582,A -85,B 0,C 180,E1 -18565.084,E2 -18565.084} C_VEL
LIN {X 0,Y 256.08,Z 318.571,A -85,B 0,C 180,E1 -18568.568,E2 -18568.568} C_VEL
LIN {X 0,Y 256.066,Z 318.561,A -85,B 0,C 180,E1 -18571.695,E2 -18571.695} C_VEL
LIN {X 0,Y 256.083,Z 318.577,A -85,B 0,C 180,E1 -18575.193,E2 -18575.193} C_VEL
LIN {X 0,Y 256.048,Z 318.588,A -85,B 0,C 180,E1 -18579.147,E2 -18579.147} C_VEL
LIN {X 0,Y 256.004,Z 318.59,A -85,B 0,C 180,E1 -18583.34,E2 -18583.34} C_VEL
LIN {X 0,Y 256.006,Z 318.597,A -85,B 0,C 180,E1 -18586.658,E2 -18586.658} C_VEL
LIN {X 0,Y 256.048,Z 318.591,A -85,B 0,C 180,E1 -18590.85,E2 -18590.85} C_VEL
LIN {X 0,Y 256.079,Z 318.586,A -85,B 0,C 180,E1 -18594.803,E2 -18594.803} C_VEL
LIN {X 0,Y 256.078,Z 318.589,A -85,B 0,C 180,E1 -18598.567,E2 -18598.567} C_VEL
LIN {X 0,Y 256.093,Z 318.584,A -85,B 0,C 180,E1 -18602.187,E2 -18602.187} C_VEL
LIN {X 0,Y 256.139,Z 318.577,A -85,B 0,C 180,E1 -18605.693,E2 -18605.693} C_VEL
LIN {X 0,Y 256.131,Z 318.584,A -85,B 0,C 180,E1 -18609.098,E2 -18609.098} C_VEL
LIN {X 0,Y 256.237,Z 318.565,A -85,B 0,C 180,E1 -18614.077,E2 -18614.077} C_VEL
LIN {X 0,Y 256.296,Z 318.558,A -85,B 0,C 180,E1 -18618.929,E2 -18618.929} C_VEL
LIN {X 0,Y 256.473,Z 318.535,A -85,B 0,C 180,E1 -18622.12,E2 -18622.12} C_VEL
LIN {X 0,Y 256.453,Z 318.54,A -85,B 0,C 180,E1 -18626.853,E2 -18626.853} C_VEL
LIN {X 0,Y 256.702,Z 318.506,A -85,B 0,C 180,E1 -18628.426,E2 -18628.426} C_VEL
LIN {X 0,Y 256.646,Z 318.612,A -85,B 0,C 180,E1 -18631.961,E2 -18631.961} C_VEL
LIN {X 0,Y 266.462,Z 343.69,A -85,B 0,C 180,E1 -18633.798,E2 -18633.798} C_VEL
LIN {X 0,Y 270.43,Z 355.009,A -85,B 0,C 180,E1 -18634.523,E2 -18634.523} C_VEL
LIN {X 0,Y 267.871,Z 426.533,A -85,B 0,C 180,E1 -18636.539,E2 -18636.539} C_VEL
LIN {X 0,Y 267.008,Z 439.945,A -85,B 0,C 180,E1 -18637.224,E2 -18637.224} C_VEL
LIN {X 0,Y 265.916,Z 452.388,A -85,B 0,C 180,E1 -18638.161,E2 -18638.161} C_VEL
LIN {X 0,Y 264.487,Z 464.361,A -85,B 0,C 180,E1 -18639.383,E2 -18639.383} C_VEL
LIN {X 0,Y 262.881,Z 475.097,A -85,B 0,C 180,E1 -18640.78,E2 -18640.78} C_VEL
LIN {X 0,Y 261.248,Z 485.172,A -85,B 0,C 180,E1 -18642.422,E2 -18642.422} C_VEL
LIN {X 0,Y 259.855,Z 493.452,A -85,B 0,C 180,E1 -18644.082,E2 -18644.082} C_VEL
LIN {X 0,Y 258.309,Z 502.049,A -85,B 0,C 180,E1 -18646.187,E2 -18646.187} C_VEL
LIN {X 0,Y 257.058,Z 509.074,A -85,B 0,C 180,E1 -18648.319,E2 -18648.319} C_VEL
LIN {X 0,Y 255.877,Z 515.968,A -85,B 0,C 180,E1 -18650.955,E2 -18650.955} C_VEL
LIN {X 0,Y 255.013,Z 521.19,A -85,B 0,C 180,E1 -18653.546,E2 -18653.546} C_VEL
LIN {X 0,Y 254.335,Z 525.157,A -85,B 0,C 180,E1 -18656.232,E2 -18656.232} C_VEL
LIN {X 0,Y 253.984,Z 527.097,A -85,B 0,C 180,E1 -18658.053,E2 -18658.053} C_VEL
LIN {X 0,Y 253.738,Z 529.021,A -85,B 0,C 180,E1 -18660.836,E2 -18660.836} C_VEL
LIN {X 0,Y 253.815,Z 529.683,A -85,B 0,C 180,E1 -18663.83,E2 -18663.83} C_VEL
LIN {X 0,Y 254.174,Z 528.981,A -85,B 0,C 180,E1 -18666.692,E2 -18666.692} C_VEL
LIN {X 0,Y 254.86,Z 527.068,A -85,B 0,C 180,E1 -18669.455,E2 -18669.455} C_VEL
LIN {X 0,Y 255.865,Z 523.991,A -85,B 0,C 180,E1 -18672.13,E2 -18672.13} C_VEL
LIN {X 0,Y 257.067,Z 519.794,A -85,B 0,C 180,E1 -18674.698,E2 -18674.698} C_VEL
LIN {X 0,Y 258.676,Z 514.277,A -85,B 0,C 180,E1 -18677.216,E2 -18677.216} C_VEL
LIN {X 0,Y 260.759,Z 507.248,A -85,B 0,C 180,E1 -18679.695,E2 -18679.695} C_VEL
LIN {X 0,Y 262.896,Z 499.595,A -85,B 0,C 180,E1 -18681.837,E2 -18681.837} C_VEL
LIN {X 0,Y 264.97,Z 491.555,A -85,B 0,C 180,E1 -18683.66,E2 -18683.66} C_VEL
LIN {X 0,Y 267.025,Z 482.624,A -85,B 0,C 180,E1 -18685.32,E2 -18685.32} C_VEL
LIN {X 0,Y 269.33,Z 472.021,A -85,B 0,C 180,E1 -18686.879,E2 -18686.879} C_VEL
LIN {X 0,Y 271.455,Z 459.882,A -85,B 0,C 180,E1 -18688.285,E2 -18688.285} C_VEL
LIN {X 0,Y 273.191,Z 447.523,A -85,B 0,C 180,E1 -18689.361,E2 -18689.361} C_VEL
LIN {X 0,Y 274.481,Z 434.192,A -85,B 0,C 180,E1 -18690.188,E2 -18690.188} C_VEL
LIN {X 0,Y 275.436,Z 421.045,A -85,B 0,C 180,E1 -18690.683,E2 -18690.683} C_VEL
LIN {X 0,Y 278.01,Z 361.014,A -85,B 0,C 180,E1 -18692.356,E2 -18692.356} C_VEL
LIN {X 0,Y 271.081,Z 345.405,A -85,B 0,C 180,E1 -18693.994,E2 -18693.994} C_VEL
LIN {X 0,Y 263.965,Z 332.186,A -85,B 0,C 180,E1 -18695.725,E2 -18695.725} C_VEL
LIN {X 0,Y 258.808,Z 323.826,A -85,B 0,C 180,E1 -18697.039,E2 -18697.039} C_VEL
LIN {X 0,Y 256.501,Z 320.247,A -85,B 0,C 180,E1 -18697.651,E2 -18697.651} C_VEL
LIN {X 0,Y 256.272,Z 319.596,A -85,B 0,C 180,E1 -18697.838,E2 -18697.838} C_VEL
LIN {X 0,Y 256.072,Z 318.593,A -85,B 0,C 180,E1 -18698.349,E2 -18698.349} C_VEL
LIN {X 0,Y 256.158,Z 318.582,A -85,B 0,C 180,E1 -18702.434,E2 -18702.434} C_VEL
LIN {X 0,Y 256.199,Z 318.571,A -85,B 0,C 180,E1 -18705.707,E2 -18705.707} C_VEL
LIN {X 0,Y 256.269,Z 318.556,A -85,B 0,C 180,E1 -18709.542,E2 -18709.542} C_VEL
LIN {X 0,Y 255.988,Z 318.595,A -85,B 0,C 180,E1 -18710.42,E2 -18710.42} C_VEL
LIN {X 0,Y 254.051,Z 318.836,A -85,B 0,C 180,E1 -18712.144,E2 -18712.144} C_VEL
LIN {X 0,Y 250.34,Z 319.3,A -85,B 0,C 180,E1 -18714.737,E2 -18714.737} C_VEL
LIN {X 0,Y 249.389,Z 319.411,A -85,B 0,C 180,E1 -18716.089,E2 -18716.089} C_VEL
LIN {X 0,Y 249.36,Z 319.415,A -85,B 0,C 180,E1 -18716.547,E2 -18716.547} C_VEL
LIN {X 0,Y 249.633,Z 319.388,A -85,B 0,C 180,E1 -18718.387,E2 -18718.387} C_VEL
LIN {X 0,Y 249.634,Z 319.389,A -85,B 0,C 180,E1 -18721.613,E2 -18721.613} C_VEL
LIN {X 0,Y 249.415,Z 319.414,A -85,B 0,C 180,E1 -18726.472,E2 -18726.472} C_VEL
LIN {X 0,Y 249.347,Z 319.426,A -85,B 0,C 180,E1 -18729.736,E2 -18729.736} C_VEL
LIN {X 0,Y 249.148,Z 319.449,A -85,B 0,C 180,E1 -18734.707,E2 -18734.707} C_VEL
LIN {X 0,Y 249.105,Z 319.452,A -85,B 0,C 180,E1 -18738.08,E2 -18738.08} C_VEL
LIN {X 0,Y 249.104,Z 319.445,A -85,B 0,C 180,E1 -18741.517,E2 -18741.517} C_VEL
LIN {X 0,Y 249.1,Z 319.446,A -85,B 0,C 180,E1 -18745.487,E2 -18745.487} C_VEL
LIN {X 0,Y 249.047,Z 319.453,A -85,B 0,C 180,E1 -18748.996,E2 -18748.996} C_VEL
LIN {X 0,Y 249.004,Z 319.461,A -85,B 0,C 180,E1 -18752.43,E2 -18752.43} C_VEL
LIN {X 0,Y 249.054,Z 319.461,A -85,B 0,C 180,E1 -18756.341,E2 -18756.341} C_VEL
LIN {X 0,Y 249.077,Z 319.46,A -85,B 0,C 180,E1 -18760.464,E2 -18760.464} C_VEL
LIN {X 0,Y 249.038,Z 319.472,A -85,B 0,C 180,E1 -18764.871,E2 -18764.871} C_VEL
LIN {X 0,Y 249.1,Z 319.614,A -85,B 0,C 180,E1 -18767.185,E2 -18767.185} C_VEL
LIN {X 0,Y 251.336,Z 327.149,A -85,B 0,C 180,E1 -18770.914,E2 -18770.914} C_VEL
LIN {X 0,Y 253.027,Z 333.197,A -85,B 0,C 180,E1 -18773.658,E2 -18773.658} C_VEL
LIN {X 0,Y 255.712,Z 338.142,A -85,B 0,C 180,E1 -18774.416,E2 -18774.416} C_VEL
LIN {X 0,Y 262.684,Z 351.948,A -85,B 0,C 180,E1 -18776.295,E2 -18776.295} C_VEL
LIN {X 0,Y 267.724,Z 363.484,A -85,B 0,C 180,E1 -18777.602,E2 -18777.602} C_VEL
LIN {X 0,Y 270.363,Z 380.637,A -85,B 0,C 180,E1 -18778.648,E2 -18778.648} C_VEL
LIN {X 0,Y 271.188,Z 388.722,A -85,B 0,C 180,E1 -18779.063,E2 -18779.063} C_VEL
LIN {X 0,Y 268.559,Z 444.263,A -85,B 0,C 180,E1 -18780.677,E2 -18780.677} C_VEL
LIN {X 0,Y 267.142,Z 458.144,A -85,B 0,C 180,E1 -18781.368,E2 -18781.368} C_VEL
LIN {X 0,Y 265.463,Z 469.569,A -85,B 0,C 180,E1 -18782.193,E2 -18782.193} C_VEL
LIN {X 0,Y 263.116,Z 482.162,A -85,B 0,C 180,E1 -18783.43,E2 -18783.43} C_VEL
LIN {X 0,Y 260.717,Z 493.421,A -85,B 0,C 180,E1 -18784.884,E2 -18784.884} C_VEL
LIN {X 0,Y 258.248,Z 503.638,A -85,B 0,C 180,E1 -18786.554,E2 -18786.554} C_VEL
LIN {X 0,Y 255.594,Z 513.676,A -85,B 0,C 180,E1 -18788.641,E2 -18788.641} C_VEL
LIN {X 0,Y 253.233,Z 522.548,A -85,B 0,C 180,E1 -18790.975,E2 -18790.975} C_VEL
LIN {X 0,Y 251.212,Z 529.698,A -85,B 0,C 180,E1 -18793.343,E2 -18793.343} C_VEL
LIN {X 0,Y 249.217,Z 536.257,A -85,B 0,C 180,E1 -18796.137,E2 -18796.137} C_VEL
LIN {X 0,Y 248.123,Z 540.619,A -85,B 0,C 180,E1 -18798.57,E2 -18798.57} C_VEL
LIN {X 0,Y 247.613,Z 542.951,A -85,B 0,C 180,E1 -18800.201,E2 -18800.201} C_VEL
LIN {X 0,Y 247.254,Z 544.839,A -85,B 0,C 180,E1 -18801.835,E2 -18801.835} C_VEL
LIN {X 0,Y 246.881,Z 547.305,A -85,B 0,C 180,E1 -18805.107,E2 -18805.107} C_VEL
LIN {X 0,Y 246.897,Z 547.952,A -85,B 0,C 180,E1 -18806.742,E2 -18806.742} C_VEL
LIN {X 0,Y 246.998,Z 548.19,A -85,B 0,C 180,E1 -18808.375,E2 -18808.375} C_VEL
LIN {X 0,Y 247.029,Z 547.989,A -85,B 0,C 180,E1 -18810.005,E2 -18810.005} C_VEL
LIN {X 0,Y 247.011,Z 547.389,A -85,B 0,C 180,E1 -18811.636,E2 -18811.636} C_VEL
LIN {X 0,Y 246.941,Z 546.385,A -85,B 0,C 180,E1 -18813.268,E2 -18813.268} C_VEL
LIN {X 0,Y 246.953,Z 544.743,A -85,B 0,C 180,E1 -18815.086,E2 -18815.086} C_VEL
LIN {X 0,Y 247.256,Z 540.682,A -85,B 0,C 180,E1 -18818.175,E2 -18818.175} C_VEL
LIN {X 0,Y 247.743,Z 536.206,A -85,B 0,C 180,E1 -18820.63,E2 -18820.63} C_VEL
LIN {X 0,Y 248.573,Z 530.495,A -85,B 0,C 180,E1 -18823.077,E2 -18823.077} C_VEL
LIN {X 0,Y 249.909,Z 523.323,A -85,B 0,C 180,E1 -18825.5,E2 -18825.5} C_VEL
LIN {X 0,Y 251.545,Z 514.347,A -85,B 0,C 180,E1 -18827.903,E2 -18827.903} C_VEL
LIN {X 0,Y 253.13,Z 505.121,A -85,B 0,C 180,E1 -18829.888,E2 -18829.888} C_VEL
LIN {X 0,Y 254.944,Z 494.907,A -85,B 0,C 180,E1 -18831.64,E2 -18831.64} C_VEL
LIN {X 0,Y 256.765,Z 483.577,A -85,B 0,C 180,E1 -18833.174,E2 -18833.174} C_VEL
LIN {X 0,Y 258.401,Z 471.876,A -85,B 0,C 180,E1 -18834.402,E2 -18834.402} C_VEL
LIN {X 0,Y 259.835,Z 459.226,A -85,B 0,C 180,E1 -18835.379,E2 -18835.379} C_VEL
LIN {X 0,Y 260.922,Z 446.018,A -85,B 0,C 180,E1 -18836.068,E2 -18836.068} C_VEL
LIN {X 0,Y 262.264,Z 411.274,A -85,B 0,C 180,E1 -18837.104,E2 -18837.104} C_VEL
LIN {X 0,Y 262.978,Z 385.501,A -85,B 0,C 180,E1 -18837.853,E2 -18837.853} C_VEL
LIN {X 0,Y 258.799,Z 355.033,A -85,B 0,C 180,E1 -18839.24,E2 -18839.24} C_VEL
LIN {X 0,Y 257.76,Z 349.495,A -85,B 0,C 180,E1 -18839.528,E2 -18839.528} C_VEL
LIN {X 0,Y 252.633,Z 335.852,A -85,B 0,C 180,E1 -18840.553,E2 -18840.553} C_VEL
LIN {X 0,Y 250.645,Z 326.382,A -85,B 0,C 180,E1 -18844.114,E2 -18844.114} C_VEL
LIN {X 0,Y 249.117,Z 319.451,A -85,B 0,C 180,E1 -18846.901,E2 -18846.901} C_VEL
LIN {X 0,Y 249.014,Z 319.471,A -85,B 0,C 180,E1 -18850.48,E2 -18850.48} C_VEL
LIN {X 0,Y 248.993,Z 319.473,A -85,B 0,C 180,E1 -18854.885,E2 -18854.885} C_VEL
LIN {X 0,Y 249.016,Z 319.467,A -85,B 0,C 180,E1 -18857.363,E2 -18857.363} C_VEL
LIN {X 0,Y 249.048,Z 319.463,A -85,B 0,C 180,E1 -18862.202,E2 -18862.202} C_VEL
LIN {X 0,Y 249.049,Z 319.46,A -85,B 0,C 180,E1 -18865.64,E2 -18865.64} C_VEL
LIN {X 0,Y 249.047,Z 319.459,A -85,B 0,C 180,E1 -18869.472,E2 -18869.472} C_VEL
LIN {X 0,Y 249.073,Z 319.458,A -85,B 0,C 180,E1 -18873.162,E2 -18873.162} C_VEL
LIN {X 0,Y 249.062,Z 319.46,A -85,B 0,C 180,E1 -18876.731,E2 -18876.731} C_VEL
LIN {X 0,Y 249.062,Z 319.455,A -85,B 0,C 180,E1 -18880.208,E2 -18880.208} C_VEL
LIN {X 0,Y 249.164,Z 319.428,A -85,B 0,C 180,E1 -18883.617,E2 -18883.617} C_VEL
LIN {X 0,Y 249.234,Z 319.436,A -85,B 0,C 180,E1 -18888.616,E2 -18888.616} C_VEL
LIN {X 0,Y 249.453,Z 319.408,A -85,B 0,C 180,E1 -18891.902,E2 -18891.902} C_VEL
LIN {X 0,Y 249.288,Z 319.419,A -85,B 0,C 180,E1 -18895.148,E2 -18895.148} C_VEL
LIN {X 0,Y 249.675,Z 319.358,A -85,B 0,C 180,E1 -18898.387,E2 -18898.387} C_VEL
LIN {X 0,Y 249.674,Z 319.375,A -85,B 0,C 180,E1 -18901.613,E2 -18901.613} C_VEL
LIN {X 0,Y 249.421,Z 319.413,A -85,B 0,C 180,E1 -18906.534,E2 -18906.534} C_VEL
LIN {X 0,Y 249.337,Z 319.421,A -85,B 0,C 180,E1 -18909.737,E2 -18909.737} C_VEL
LIN {X 0,Y 249.174,Z 319.444,A -85,B 0,C 180,E1 -18914.705,E2 -18914.705} C_VEL
LIN {X 0,Y 249.089,Z 319.45,A -85,B 0,C 180,E1 -18918.081,E2 -18918.081} C_VEL
LIN {X 0,Y 249.048,Z 319.459,A -85,B 0,C 180,E1 -18921.522,E2 -18921.522} C_VEL
LIN {X 0,Y 249.043,Z 319.459,A -85,B 0,C 180,E1 -18925.436,E2 -18925.436} C_VEL
LIN {X 0,Y 249.028,Z 319.447,A -85,B 0,C 180,E1 -18928.966,E2 -18928.966} C_VEL
LIN {X 0,Y 249.001,Z 319.444,A -85,B 0,C 180,E1 -18932.43,E2 -18932.43} C_VEL
LIN {X 0,Y 249.017,Z 319.462,A -85,B 0,C 180,E1 -18936.348,E2 -18936.348} C_VEL
LIN {X 0,Y 248.977,Z 319.471,A -85,B 0,C 180,E1 -18940.484,E2 -18940.484} C_VEL
LIN {X 0,Y 248.966,Z 319.473,A -85,B 0,C 180,E1 -18944.888,E2 -18944.888} C_VEL
LIN {X 0,Y 248.974,Z 319.469,A -85,B 0,C 180,E1 -18947.35,E2 -18947.35} C_VEL
LIN {X 0,Y 249.009,Z 319.466,A -85,B 0,C 180,E1 -18951.613,E2 -18951.613} C_VEL
LIN {X 0,Y 249.048,Z 319.458,A -85,B 0,C 180,E1 -18955.636,E2 -18955.636} C_VEL
LIN {X 0,Y 248.998,Z 319.469,A -85,B 0,C 180,E1 -18959.462,E2 -18959.462} C_VEL
LIN {X 0,Y 249.037,Z 319.468,A -85,B 0,C 180,E1 -18963.154,E2 -18963.154} C_VEL
LIN {X 0,Y 249.059,Z 319.461,A -85,B 0,C 180,E1 -18966.727,E2 -18966.727} C_VEL
LIN {X 0,Y 249.065,Z 319.459,A -85,B 0,C 180,E1 -18970.204,E2 -18970.204} C_VEL
LIN {X 0,Y 249.183,Z 319.446,A -85,B 0,C 180,E1 -18973.614,E2 -18973.614} C_VEL
LIN {X 0,Y 249.239,Z 319.436,A -85,B 0,C 180,E1 -18978.611,E2 -18978.611} C_VEL
LIN {X 0,Y 249.422,Z 319.413,A -85,B 0,C 180,E1 -18981.896,E2 -18981.896} C_VEL
LIN {X 0,Y 249.264,Z 319.434,A -85,B 0,C 180,E1 -18985.143,E2 -18985.143} C_VEL
LIN {X 0,Y 249.662,Z 319.383,A -85,B 0,C 180,E1 -18988.382,E2 -18988.382} C_VEL
LIN {X 0,Y 249.644,Z 319.387,A -85,B 0,C 180,E1 -18991.205,E2 -18991.205} C_VEL
LIN {X 0,Y 250.769,Z 322.413,A -85,B 0,C 180,E1 -18991.469,E2 -18991.469} C_VEL
LIN {X 0,Y 260.207,Z 345.891,A -85,B 0,C 180,E1 -18993.249,E2 -18993.249} C_VEL
LIN {X 0,Y 263.894,Z 356.794,A -85,B 0,C 180,E1 -18993.962,E2 -18993.962} C_VEL
LIN {X 0,Y 261.275,Z 426.969,A -85,B 0,C 180,E1 -18995.991,E2 -18995.991} C_VEL
LIN {X 0,Y 260.306,Z 440.947,A -85,B 0,C 180,E1 -18996.729,E2 -18996.729} C_VEL
LIN {X 0,Y 259.208,Z 453.112,A -85,B 0,C 180,E1 -18997.688,E2 -18997.688} C_VEL
LIN {X 0,Y 257.615,Z 465.671,A -85,B 0,C 180,E1 -18999.019,E2 -18999.019} C_VEL
LIN {X 0,Y 255.968,Z 476.406,A -85,B 0,C 180,E1 -19000.482,E2 -19000.482} C_VEL
LIN {X 0,Y 254.285,Z 486.258,A -85,B 0,C 180,E1 -19002.16,E2 -19002.16} C_VEL
LIN {X 0,Y 252.562,Z 495.973,A -85,B 0,C 180,E1 -19004.238,E2 -19004.238} C_VEL
LIN {X 0,Y 251.138,Z 503.599,A -85,B 0,C 180,E1 -19006.244,E2 -19006.244} C_VEL
LIN {X 0,Y 249.641,Z 511.653,A -85,B 0,C 180,E1 -19008.883,E2 -19008.883} C_VEL
LIN {X 0,Y 248.513,Z 517.941,A -85,B 0,C 180,E1 -19011.563,E2 -19011.563} C_VEL
LIN {X 0,Y 247.81,Z 522.446,A -85,B 0,C 180,E1 -19014.054,E2 -19014.054} C_VEL
LIN {X 0,Y 247.069,Z 526.408,A -85,B 0,C 180,E1 -19017.065,E2 -19017.065} C_VEL
LIN {X 0,Y 246.77,Z 528.094,A -85,B 0,C 180,E1 -19018.949,E2 -19018.949} C_VEL
LIN {X 0,Y 246.662,Z 529.437,A -85,B 0,C 180,E1 -19021.265,E2 -19021.265} C_VEL
LIN {X 0,Y 246.77,Z 529.93,A -85,B 0,C 180,E1 -19024.318,E2 -19024.318} C_VEL
LIN {X 0,Y 247.198,Z 529.114,A -85,B 0,C 180,E1 -19027.244,E2 -19027.244} C_VEL
LIN {X 0,Y 247.96,Z 527.099,A -85,B 0,C 180,E1 -19030.069,E2 -19030.069} C_VEL
